// TIA Portal project "Voltra_Nord" (V21)

(* hardware
DEVICE "ET 200SP station_1"  ET 200SP-Station
   slot 0: "Rack_0"  Rack  6ES5 710-8MAx1
   slot 1: "Volta_Nord"  CPU 1510SP-1 PN  6ES7 510-1DK03-0AB0  V4.0
      slot 32768: "PROFINET interface_1"  X1
         slot 32771: "Port_3"  X1 P3
   slot 2: "CM PtP_1"  CM PtP  6ES7 137-6AA01-0BA0  V2.0
      slot 1: "CM PtP_1"  CM PtP Sub
   slot 3: "AI 8xRTD/TC 2-wire HF_1"  AI 8xRTD/TC 2-wire HF  6ES7 134-6JF00-0CA1  V2.1
      slot 1: "AI 8xRTD/TC 2-wire HF_1"  AI 8xRTD/TC 2-wire HF
   slot 4: "AI 8xRTD/TC 2-wire HF_2"  AI 8xRTD/TC 2-wire HF  6ES7 134-6JF00-0CA1  V2.1
      slot 1: "AI 8xRTD/TC 2-wire HF_2"  AI 8xRTD/TC 2-wire HF
   slot 5: "AI 8xI 2-/4-wire BA_1"  AI 8xI 2-,4-wire BA  6ES7 134-6GF00-0AA1  V1.0
      slot 1: "AI 8xI 2-/4-wire BA_1"  AI 8xI 2-,4-wire BA
   slot 6: "AI 8xI 2-/4-wire BA_2"  AI 8xI 2-,4-wire BA  6ES7 134-6GF00-0AA1  V1.0
      slot 1: "AI 8xI 2-/4-wire BA_2"  AI 8xI 2-,4-wire BA
   slot 7: "AQ 4xU/I ST_1"  AQ 4xU/I ST  6ES7 135-6HD00-0BA1  V1.1
      slot 1: "AQ 4xU/I ST_1"  AQ 4xU/I ST
   slot 8: "DI 16x24VDC ST_1"  DI 16x24VDC ST  6ES7 131-6BH01-0BA0  V0.0
      slot 1: "DI 16x24VDC ST_1"  DI 16x24VDC ST
   slot 9: "DI 16x24VDC ST_2"  DI 16x24VDC ST  6ES7 131-6BH01-0BA0  V0.0
      slot 1: "DI 16x24VDC ST_2"  DI 16x24VDC ST
   slot 10: "DI 16x24VDC ST_3"  DI 16x24VDC ST  6ES7 131-6BH01-0BA0  V0.0
      slot 1: "DI 16x24VDC ST_3"  DI 16x24VDC ST
   slot 11: "DQ 16x24VDC/0.5A BA_1"  DQ 16x24VDC/0.5A BA  6ES7 132-6BH00-0AA0  V0.0
      slot 1: "DQ 16x24VDC/0.5A BA_1"  DQ 16x24VDC/0.5A BA
   slot 12: "DQ 16x24VDC/0.5A BA_2"  DQ 16x24VDC/0.5A BA  6ES7 132-6BH00-0AA0  V0.0
      slot 1: "DQ 16x24VDC/0.5A BA_2"  DQ 16x24VDC/0.5A BA
   slot 13: "DQ 16x24VDC/0.5A BA_3"  DQ 16x24VDC/0.5A BA  6ES7 132-6BH00-0AA0  V0.0
      slot 1: "DQ 16x24VDC/0.5A BA_3"  DQ 16x24VDC/0.5A BA
   slot 14: "Server module_1"  Server module  6ES7 193-6PA00-0AA0  V1.2
      slot 1: "Server module_1"  Server module
   slot 127: "BA 2xRJ45"  BA 2xRJ45  6ES7 193-6AR00-0AA0  V0.0
      slot 32769: "Port_1"  X1 P1  6ES7 193-6AR00-0AA0
      slot 32770: "Port_2"  X1 P2  6ES7 193-6AR00-0AA0
*)

// ===== PLC "Volta_Nord"  CPU 1510SP-1 PN =====

VAR_GLOBAL   // PLC tag table "Default tag table"
   "Tag_1" AT %M100.0 : Bool;
   "System_Byte" AT %MB1 : Byte;
   "FirstScan" AT %M1.0 : Bool;
   "DiagStatusUpdate" AT %M1.1 : Bool;
   "AlwaysTRUE" AT %M1.2 : Bool;
   "AlwaysFALSE" AT %M1.3 : Bool;
   "Clock_Byte" AT %MB0 : Byte;
   "Clock_10Hz" AT %M0.0 : Bool;
   "Clock_5Hz" AT %M0.1 : Bool;
   "Clock_2.5Hz" AT %M0.2 : Bool;
   "Clock_2Hz" AT %M0.3 : Bool;
   "Clock_1.25Hz" AT %M0.4 : Bool;
   "Clock_1Hz" AT %M0.5 : Bool;
   "Clock_0.625Hz" AT %M0.6 : Bool;
   "Clock_0.5Hz" AT %M0.7 : Bool;
END_VAR

VAR_GLOBAL   // PLC tag table "RTD"
   "rM1OilTemp_C" AT %IW8 : Int;
   "rM1SuctionTemp_C" AT %IW10 : Int;
   "rM1DischargeTemp_C" AT %IW12 : Int;
   "rM2OilTemp_C" AT %IW14 : Int;
   "rM2SuctionTemp_C" AT %IW16 : Int;
   "rM2DischargeTemp_C" AT %IW18 : Int;
   "rM1EvapWaterOutTemp_C" AT %IW24 : Int;
   "rM1EvapWaterInTemp_C" AT %IW26 : Int;
   "rM1CondWaterOutTemp_C" AT %IW28 : Int;
   "rM1CondWaterInTemp_C" AT %IW30 : Int;
   "rM2EvapWaterOutTemp_C" AT %IW32 : Int;
   "rM2EvapWaterInTemp_C" AT %IW34 : Int;
   "rM2CondWaterOutTemp_C" AT %IW36 : Int;
   "rM2CondWaterInTemp_C" AT %IW38 : Int;
   "rm1OilTemp2_C" AT %IW20 : Int;
   "rm2OilTemp2_C" AT %IW22 : Int;
END_VAR

VAR_GLOBAL   // PLC tag table "AI"
   "rM1LiquidLevel_pct" AT %IW40 : Int;
   "rM1Pdis_bar" AT %IW42 : Int;
   "rM1Psuc_bar" AT %IW44 : Int;
   "rM1ViValvePos_pct" AT %IW46 : Int;
   "rM1ExtSetpointInput_C" AT %IW48 : Int;   // 9-10 klemes
   "rM2LiquidLevel_pct" AT %IW50 : Int;
   "rM2Pdis_bar" AT %IW52 : Int;
   "rM2Psuc_bar" AT %IW54 : Int;
   "rM2ExtSetpointInput_C" AT %IW58 : Int;   // 19-20 klemens
   "rM2ViValvePos_pct" AT %IW56 : Int;
   "AI_Rezerve1" AT %IW60 : Int;
   "AI_Rezerve2" AT %IW62 : Int;
   "AI_Rezerve3" AT %IW64 : Int;
   "AI_Rezerve4" AT %IW66 : Int;
   "AI_Rezerve5" AT %IW68 : Int;
   "AI_Rezerve6" AT %IW70 : Int;
END_VAR

VAR_GLOBAL   // PLC tag table "AQ"
   "rM1CompFreqRefOut_Hz" AT %QW0 : Int;
   "rM1ViValveCmd_pct" AT %QW2 : Int;
   "rM2CompFreqRefOut_Hz" AT %QW4 : Int;
   "rM2ViValveCmd_pct" AT %QW6 : Int;
END_VAR

VAR_GLOBAL   // PLC tag table "DI"
   "xPhaseProtectionRelaySig" AT %I72.0 : Bool;
   "xSafetySignal" AT %I72.1 : Bool;
   "xEmgStop" AT %I72.2 : Bool;
   "xM1EvapMotRunning" AT %I72.3 : Bool;
   "xM1CondenserMotRunning" AT %I72.4 : Bool;
   "xM1ExhaustFanRunning" AT %I72.5 : Bool;
   "xM1CompDriverRunnig" AT %I72.6 : Bool;
   "xM1CompDriverFault" AT %I72.7 : Bool;
   "xM1LiquidLowLevelSw" AT %I73.0 : Bool;
   "xM1LiquidHighLevelSw" AT %I73.1 : Bool;
   "xM2EvapMotRunning" AT %I73.2 : Bool;
   "xM2CondenserMotRunning" AT %I73.3 : Bool;
   "xM2ExhaustFanRunning" AT %I73.4 : Bool;
   "xM2CompDriverRunnig" AT %I73.5 : Bool;
   "xM2CompDriverFault" AT %I73.6 : Bool;
   "xM2LiquidLowLevelSw" AT %I73.7 : Bool;
   "xM2LiquidHighLevelSw" AT %I74.0 : Bool;
   "xM1OilFlowSw" AT %I74.1 : Bool;
   "xM1HighPressureSw" AT %I74.2 : Bool;
   "xM1LowPressureSw" AT %I74.3 : Bool;
   "xM1OilTankLowLevelSw" AT %I74.4 : Bool;
   "xM2OilFlowSw" AT %I74.5 : Bool;
   "xM2HighPressureSw" AT %I74.6 : Bool;
   "xM2LowPressureSw" AT %I74.7 : Bool;
   "xM2OilTankLowLevelSw" AT %I75.0 : Bool;
   "xM1BmsStartCoolEnableIn" AT %I75.1 : Bool;
   "xM1BmsStartHeatEnableIn" AT %I75.2 : Bool;
   "xM2BmsStartCoolEnableIn" AT %I75.3 : Bool;
   "xM2BmsStartHeatEnableIn" AT %I75.4 : Bool;
   "xM1EvapFlowSw" AT %I75.5 : Bool;
   "xM2EvapFlowSw" AT %I75.6 : Bool;
   "xM1CondenFlowSw" AT %I75.7 : Bool;
   "xM2CondenFlowSw" AT %I76.0 : Bool;
   "xM1OilHighLevelSwitch" AT %I76.1 : Bool;
   "xM2OilHighLevelSwitch" AT %I76.2 : Bool;
   "xM1GasFault" AT %I76.3 : Bool;
   "xM2GasFault" AT %I76.4 : Bool;
   "xM1CompThermalFault" AT %I76.5 : Bool;
   "xM2CompThermalFault" AT %I76.6 : Bool;
   "xM1HeaterRunnig" AT %I76.7 : Bool;
   "xM2HeaterRunnig" AT %I77.0 : Bool;
   "DI_Rezerve3" AT %I77.1 : Bool;
   "DI_Rezerve4" AT %I77.2 : Bool;
   "DI_Rezerve5" AT %I77.3 : Bool;
   "DI_Rezerve6" AT %I77.4 : Bool;
   "DI_Rezerve7" AT %I77.5 : Bool;
   "DI_Rezerve8" AT %I77.6 : Bool;
   "DI_Rezerve9" AT %I77.7 : Bool;
END_VAR

VAR_GLOBAL   // PLC tag table "DQ"
   "xM1EvapPumpCmd" AT %Q8.0 : Bool;
   "xM1CondPumpCmd" AT %Q8.1 : Bool;
   "xM1ExhaustFanCmd" AT %Q8.2 : Bool;
   "xM1CompRunCmd" AT %Q8.3 : Bool;
   "xM1TwoWayValveCmd" AT %Q8.4 : Bool;
   "xM1MvsEnableCmd1" AT %Q8.5 : Bool;   // 24v dc inildi panoda
   "xM1SystemOnRelayCmd" AT %Q8.6 : Bool;
   "xM1FaultRelayCmd" AT %Q8.7 : Bool;
   "xM1OilInletSolValve1Cmd" AT %Q9.0 : Bool;
   "xM1OilITempValve" AT %Q9.1 : Bool;
   "xM1OilReturnValve1" AT %Q9.2 : Bool;
   "xM1OilReturnValve2" AT %Q9.3 : Bool;
   "xM1StartLampCmd" AT %Q9.4 : Bool;
   "xM1FaultLampCmd" AT %Q9.5 : Bool;
   "xM1StopLampCmd" AT %Q9.6 : Bool;
   "xM2EvapPumpCmd" AT %Q9.7 : Bool;
   "xM2CondPumpCmd" AT %Q10.0 : Bool;
   "xM2ExhaustFanCmd" AT %Q10.1 : Bool;
   "xM2CompRunCmd" AT %Q10.2 : Bool;
   "xM2TwoWayValveCmd" AT %Q10.3 : Bool;
   "xM2MvsEnableCmd1" AT %Q10.4 : Bool;
   "xM2SystemOnRelayCmd" AT %Q10.5 : Bool;
   "xM2FaultRelayCmd" AT %Q10.6 : Bool;
   "xM2OillInletSolValve1Cmd" AT %Q10.7 : Bool;
   "xM2OilITempValve" AT %Q11.0 : Bool;
   "xM2OilReturnValve1" AT %Q11.1 : Bool;
   "xM2OilReturnValve2" AT %Q11.2 : Bool;
   "xM2StartLampCmd" AT %Q11.3 : Bool;
   "xM2FaultLampCmd" AT %Q11.4 : Bool;
   "xM2StopLampCmd" AT %Q11.5 : Bool;
   "xM1OilFlowValve" AT %Q11.6 : Bool;   // ICFE20H Slenoid Valve
   "xM2OilFlowValve" AT %Q11.7 : Bool;   // ICFE20H Slenoid Valve
   "xM1OilHeater" AT %Q12.0 : Bool;
   "xM2OilHeater" AT %Q12.1 : Bool;
   "xM1MvsEnableCmd2" AT %Q12.2 : Bool;
   "xM2MvsEnableCmd2" AT %Q12.3 : Bool;
   "DQ_Rezerve1" AT %Q12.4 : Bool;   // 220V AC PANOYA İNİLDİ
   "DQ_Rezerve2" AT %Q12.5 : Bool;   // 220V AC PANOYA İNİLDİ
   "DQ_Rezerve3" AT %Q12.6 : Bool;   // 220V AC PANOYA İNİLDİ
   "DQ_Rezerve4" AT %Q12.7 : Bool;   // 220V AC PANOYA İNİLDİ
   "DQ_Rezerve5" AT %Q13.0 : Bool;   // KURU KONTAK İNİLDİ
   "DQ_Rezerve6" AT %Q13.1 : Bool;   // KURU KONTAK İNİLDİ
   "DQ_Rezerve7" AT %Q13.2 : Bool;
   "DQ_Rezerve8" AT %Q13.3 : Bool;
   "DQ_Rezerve9" AT %Q13.4 : Bool;
   "DQ_Rezerve10" AT %Q13.5 : Bool;
   "DQ_Rezerve11" AT %Q13.6 : Bool;
   "DQ_Rezerve12" AT %Q13.7 : Bool;
END_VAR

DATA_BLOCK "AuxOutput"   // DB24
{ S7_Optimized_Access := 'TRUE' }
VERSION : 0.1
   VAR
      m1OilTempSelenoid : Bool;   // Makine 1 5 numara yağ soğutucusunun 25 numaralı valfinin çalışması için
      m2OilTempSelenoid : Bool;   // Makine 2 5 numara yağ soğutucusunun 25 numaralı valfinin çalışması için
      m1EvapOilValve3 : Bool;   // Makine 1 24 numaralı ekipman 1. selenoid valfi
      m1EvapOilValve4 : Bool;   // Makine 1 24 numaralı ekipman 2. selenoid valfi
      m2EvapOilValve3 : Bool;
      m2EvapOilValve4 : Bool;
   END_VAR
BEGIN
END_DATA_BLOCK

DATA_BLOCK "Alarm_DB"   // DB31
{ S7_Optimized_Access := 'FALSE' }
VERSION : 0.1
   VAR
      ALM_m1DischargeHighPressure : Bool;
      ALM_m2DischargeHighPressure : Bool;
      ALM_m1DischargeLowPressure : Bool;
      ALM_m2DischargeLowPressure : Bool;
      ALM_m1KrıwanThermalFault : Bool;
      ALM_m2KrıwanThermalFault : Bool;
      ALM_m1OilFlowFault : Bool;
      ALM_m2OilFlowFault : Bool;
      ALM_m1CondensFlowFault : Bool;
      ALM_m2CondensFlowFault : Bool;
      ALM_m1EvapFlowFault : Bool;
      ALM_m2EvapFlowFault : Bool;
      ALM_m1EvapLiquidHighLevelFault : Bool;
      ALM_m2EvapLiquidHighLevelFault : Bool;
      ALM_m1EvapLiquidLowLevelFault : Bool;
      ALM_m2EvapLiquidLowLevelFault : Bool;
      ALM_m1OilTempHighFault : Bool;
      ALM_m2OilTempHighFault : Bool;
      ALM_m1OilTempHighHighFault : Bool;
      ALM_m2OilTempHighHighFault : Bool;
      ALM_m1EvapFlowWarning : Bool;
      ALM_m2EvapFlowWarning : Bool;
      ALM_m1CondensFlowWarning : Bool;
      ALM_m2CondensFlowWarning : Bool;
      ALM_m1NH3Fault : Bool;
      ALM_m2NH3Fault : Bool;
      ALM_m1CompInvFault : Bool;
      ALM_m2CompInvFault : Bool;
      ALM_PhaseProtectionRelayFault : Bool;
      ALM_SafetyFault : Bool;
      ALM_EmgFault : Bool;
      ALM_m1CompDriverFault : Bool;
      ALM_m2CompDriverFault : Bool;
      ALM_m1CondensMotorFault : Bool;
      ALM_m2CondensMotorFault_1 : Bool;
      ALM_m1EvapMotorFault : Bool;
      ALM_m2EvapMotorFault : Bool;
   END_VAR
BEGIN
END_DATA_BLOCK

DATA_BLOCK "General_DB"   // DB32
{ S7_Optimized_Access := 'FALSE' }
VERSION : 0.1
   VAR
      m1FlowOilAlarmEnable : Bool;
      m2FlowOilAlarmEnable : Bool;
      m1CondensFlowAlarmEnable : Bool;
      m2CondensFlowAlarmEnable : Bool;
      m1EvapFlowAlarmEnable : Bool;
      m2EvapFlowAlarmEnable : Bool;
      m1EvapLiquidHighLevelEnable : Bool;
      m2EvapLiquidHighLevelEnable : Bool;
      m1EvapLiquidLowLevelEnable : Bool;
      m2EvapLiquidLowLevelEnable : Bool;
      m1OilTempHighHighEnable : Bool;
      m2OilTempHighHighEnable : Bool;
      m1DischargeTempHighEnable : Bool;
      m2DischargeTempHighEnable : Bool;
      m1DischargeTempHighHighEnable : Bool;
      m2DischargeTempHighHighEnable : Bool;
      m1EvapFlowWarningEnable : Bool;
      m2EvapFlowWarningEnable : Bool;
      m1CondensFlowWarningEnable : Bool;
      m2CondensFlowWarningEnable : Bool;
      m1OilTempHighEnable : Bool;
      m2OilTempHighEnable : Bool;
      m1OilTempOk : Bool;
      m2OilTempOk : Bool;
      m1Status : Int;
      m2Status : Int;
      m1StartCoolling : Bool;
      m1StartHeating : Bool;
   END_VAR
BEGIN
END_DATA_BLOCK

DATA_BLOCK "PidVar_DB"   // DB41
{ S7_Optimized_Access := 'FALSE' }
VERSION : 0.1
   VAR
      m1PidSetPoint : Real;
      m1ManualEnable : Bool;
      m1ManualValue : Real;
      m1ErrorAck : Bool;
      m1Reset : Bool;
      m1ModeActivate : Bool;
      m1Mode : Int;
      m2PidSetPoint : Real;
      m2ManualEnable : Bool;
      m2ManualValue : Real;
      m2ErrorAck : Bool;
      m2Reset : Bool;
      m2ModeActivate : Bool;
      m2Mode : Int;
      m1LiquidLevelSet : Real;
      m1ExpManEnable : Bool;
      m1ExpManValue : Real;
      m1LiquidErrorAck : Bool;
      m1LiquidPidReset : Bool;
      m1LiquidModeActive : Bool;
      m1LiquidModePid : Int;
      m2LiquidLevelSet : Real;
      m2ExpManEnable : Bool;
      m2ExpManValue : Real;
      m2LiquidErrorAck : Bool;
      m2LiquidPidReset : Bool;
      m2LiquidModeActive : Bool;
      m2LiquidModePid : Int;
   END_VAR
BEGIN
END_DATA_BLOCK

// folder: Hmi

DATA_BLOCK "Pressure_Scale"   // DB2
{ S7_Optimized_Access := 'FALSE' }
VERSION : 0.1
   VAR
      M1PdisOut_Max : Real;
      M1PdisOut_Min : Real;
      M1PdisIn_Max : Real;
      M1PdisIn_Min : Real;
      M1PdisAlpha : Real := 1.0;
      M2PdisOut_Max : Real;
      M2PdisOut_Min : Real;
      M2PdisIn_Max : Real;
      M2PdisIn_Min : Real;
      M2PdisAlpha : Real := 1.0;
      M1PSecOut_Max : Real;
      M1PSecOut_Min : Real;
      M1PSecIn_Max : Real;
      M1PSecIn_Min : Real;
      M1PSecAlpha : Real := 1.0;
      M2PSecOut_Max : Real;
      M2PSecOut_Min : Real;
      M2PSecIn_Max : Real;
      M2PSecIn_Min : Real;
      M2PSecAlpha : Real := 1.0;
   END_VAR
BEGIN
END_DATA_BLOCK

DATA_BLOCK "Liquid_Level"   // DB6
{ S7_Optimized_Access := 'FALSE' }
VERSION : 0.1
   VAR
      M1LiquidLvlOut_Max : Real;
      M1LiquidLvlOut_Min : Real;
      M1LiquidLvlIn_Max : Real;
      M1LiquidLvlIn_Min : Real;
      M1LiquidLvlAlpha : Real;
      M2LiquidLvlOut_Max : Real;
      M2LiquidLvlOut_Min : Real;
      M2LiquidLvlIn_Max : Real;
      M2LiquidLvlIn_Min : Real;
      M2LiquidLvlAlpha : Real;
   END_VAR
BEGIN
END_DATA_BLOCK

DATA_BLOCK "HMI"   // DB23
{ S7_Optimized_Access := 'FALSE' }
VERSION : 0.1
   VAR
      rM1OilTempHis : Real;
      rM1OilTempSet : Real;
      rM2OilTempHis : Real;
      rM2OilTempSet : Real;
      tM1EvapOilHisTime : Time;   // M1 24 numaralı ekipman sensörünün filtresi için koyuldu
      tM1EvapOilDischargeTime : Time;   // M1 24 numaralı ekipmanın basınç hattının valfinin açık kalma süresi
      tM1EvapOilDischargeWaitTime : Time;   // M1 24 numaralı ekipmanın basınç hattının valfinin bekleme süresi
      tM2EvapOilHisTime : Time;
      tM2EvapOilDischargeTime : Time;
      tM2EvapOilDischargeWaitTime : Time;
      m1SetDischargeHighPressure : Real;
      m2SetDischargeHighPressure : Real;
      m1SetDischargeLowPressure : Real;
      m2SetDischargeLowPressure : Real;
      m1OilTempHighHighSet : Real;
      m2OilTempHighHighSet : Real;
      m1DischargeTempHighSet : Real;
      m2DischargeTempHighSet : Real;
      m1DischargeTempHighHighSet : Real;
      m2DischargeTempHighHighSet : Real;
      m1OilTempHighSet : Real;
      m2OilTempHighSet : Real;
      m1OilStartTempSet : Real;
      m2OilStartTempSet : Real;
      m1Status : Int;
      m1ExtValveScaleAlpha : Real := 1.0;
      m2ExtValveScaleAlpha : Real := 1.0;
   END_VAR
BEGIN
END_DATA_BLOCK

DATA_BLOCK "TempSet"   // DB39
{ S7_Optimized_Access := 'FALSE' }
VERSION : 0.1
   VAR
      m1TempSetOut_Max : Real;
      m1TempSetOut_Min : Real;
      m1TempSetIn_Max : Real;
      m1TempSetIn_Min : Real;
      m1TempSetAlpha : Real := 1.0;
      m2TempSetOut_Max : Real;
      m2TempSetOut_Min : Real;
      m2TempSetIn_Max : Real;
      m2TempSetIn_Min : Real;
      m2TempSetAlpha : Real := 1.0;
   END_VAR
BEGIN
END_DATA_BLOCK

// folder: Scale_DB

DATA_BLOCK "M1Pdischarge"   // DB1
{ S7_Optimized_Access := 'TRUE' }
VERSION : 0.1
// stored: InstanceOfName Scale
"Scale"
BEGIN
END_DATA_BLOCK

DATA_BLOCK "M2Pdischarge"   // DB3
{ S7_Optimized_Access := 'TRUE' }
VERSION : 0.1
// stored: InstanceOfName Scale
"Scale"
BEGIN
END_DATA_BLOCK

DATA_BLOCK "M1PSec"   // DB4
{ S7_Optimized_Access := 'TRUE' }
VERSION : 0.1
// stored: InstanceOfName Scale
"Scale"
BEGIN
END_DATA_BLOCK

DATA_BLOCK "M2Psec"   // DB5
{ S7_Optimized_Access := 'TRUE' }
VERSION : 0.1
// stored: InstanceOfName Scale
"Scale"
BEGIN
END_DATA_BLOCK

DATA_BLOCK "M1LiquidLevel"   // DB7
{ S7_Optimized_Access := 'TRUE' }
VERSION : 0.1
// stored: InstanceOfName Scale
"Scale"
BEGIN
END_DATA_BLOCK

DATA_BLOCK "M2LiquidLevel"   // DB8
{ S7_Optimized_Access := 'TRUE' }
VERSION : 0.1
// stored: InstanceOfName Scale
"Scale"
BEGIN
END_DATA_BLOCK

DATA_BLOCK "m1Discharge_TT"   // DB9
{ S7_Optimized_Access := 'TRUE' }
VERSION : 0.1
// stored: InstanceOfName RTD
"RTD"
BEGIN
END_DATA_BLOCK

DATA_BLOCK "m2Discharge_TT"   // DB10
{ S7_Optimized_Access := 'TRUE' }
VERSION : 0.1
// stored: InstanceOfName RTD
"RTD"
BEGIN
END_DATA_BLOCK

DATA_BLOCK "m1Section_TT"   // DB11
{ S7_Optimized_Access := 'TRUE' }
VERSION : 0.1
// stored: InstanceOfName RTD
"RTD"
BEGIN
END_DATA_BLOCK

DATA_BLOCK "m2Section_TT"   // DB12
{ S7_Optimized_Access := 'TRUE' }
VERSION : 0.1
// stored: InstanceOfName RTD
"RTD"
BEGIN
END_DATA_BLOCK

DATA_BLOCK "m1Oil_TT"   // DB13
{ S7_Optimized_Access := 'TRUE' }
VERSION : 0.1
// stored: InstanceOfName RTD
"RTD"
BEGIN
END_DATA_BLOCK

DATA_BLOCK "m2Oil_TT"   // DB14
{ S7_Optimized_Access := 'TRUE' }
VERSION : 0.1
// stored: InstanceOfName RTD
"RTD"
BEGIN
END_DATA_BLOCK

DATA_BLOCK "m1EvapWatOut_TT"   // DB15
{ S7_Optimized_Access := 'TRUE' }
VERSION : 0.1
// stored: InstanceOfName RTD
"RTD"
BEGIN
END_DATA_BLOCK

DATA_BLOCK "m1EvapWatIn_TT"   // DB16
{ S7_Optimized_Access := 'TRUE' }
VERSION : 0.1
// stored: InstanceOfName RTD
"RTD"
BEGIN
END_DATA_BLOCK

DATA_BLOCK "m2EvapWatOut_TT"   // DB17
{ S7_Optimized_Access := 'TRUE' }
VERSION : 0.1
// stored: InstanceOfName RTD
"RTD"
BEGIN
END_DATA_BLOCK

DATA_BLOCK "m2EvapWatIn_TT"   // DB18
{ S7_Optimized_Access := 'TRUE' }
VERSION : 0.1
// stored: InstanceOfName RTD
"RTD"
BEGIN
END_DATA_BLOCK

DATA_BLOCK "m1ConWatOut_TT"   // DB19
{ S7_Optimized_Access := 'TRUE' }
VERSION : 0.1
// stored: InstanceOfName RTD
"RTD"
BEGIN
END_DATA_BLOCK

DATA_BLOCK "m1ConWatIn_TT"   // DB20
{ S7_Optimized_Access := 'TRUE' }
VERSION : 0.1
// stored: InstanceOfName RTD
"RTD"
BEGIN
END_DATA_BLOCK

DATA_BLOCK "m2ConWatOut_TT"   // DB21
{ S7_Optimized_Access := 'TRUE' }
VERSION : 0.1
// stored: InstanceOfName RTD
"RTD"
BEGIN
END_DATA_BLOCK

DATA_BLOCK "m2ConWatIn_TT"   // DB22
{ S7_Optimized_Access := 'TRUE' }
VERSION : 0.1
// stored: InstanceOfName RTD
"RTD"
BEGIN
END_DATA_BLOCK

DATA_BLOCK "m1TempSetScale"   // DB38
{ S7_Optimized_Access := 'TRUE' }
VERSION : 0.1
// stored: InstanceOfName Scale
"Scale"
BEGIN
END_DATA_BLOCK

DATA_BLOCK "m2TempSetScale"   // DB40
{ S7_Optimized_Access := 'TRUE' }
VERSION : 0.1
// stored: InstanceOfName Scale
"Scale"
BEGIN
END_DATA_BLOCK

DATA_BLOCK "m1ExtValvePoz"   // DB45
{ S7_Optimized_Access := 'TRUE' }
VERSION : 0.1
// stored: InstanceOfName Scale
"Scale"
BEGIN
END_DATA_BLOCK

DATA_BLOCK "m2ExtValvePoz"   // DB46
{ S7_Optimized_Access := 'TRUE' }
VERSION : 0.1
// stored: InstanceOfName Scale
"Scale"
BEGIN
END_DATA_BLOCK

// folder: System blocks/Program resources

DATA_BLOCK "m1EvapOilSenFilter_Time"   // DB25
{ S7_Optimized_Access := 'TRUE' }
AUTHOR : Simatic
FAMILY : IEC
NAME : IEC_TMR
VERSION : 1.0
// stored: InstanceOfName IEC_TIMER
"IEC_TIMER"
BEGIN
END_DATA_BLOCK

DATA_BLOCK "m1EvapOilValve4Run_Time"   // DB26
{ S7_Optimized_Access := 'TRUE' }
AUTHOR : Simatic
FAMILY : IEC
NAME : IEC_TMR
VERSION : 1.0
// stored: InstanceOfName IEC_TIMER
"IEC_TIMER"
BEGIN
END_DATA_BLOCK

DATA_BLOCK "m1EvapOilValve4Wait_Time"   // DB27
{ S7_Optimized_Access := 'TRUE' }
AUTHOR : Simatic
FAMILY : IEC
NAME : IEC_TMR
VERSION : 1.0
// stored: InstanceOfName IEC_TIMER
"IEC_TIMER"
BEGIN
END_DATA_BLOCK

DATA_BLOCK "m2EvapOilSenFilter_Time"   // DB28
{ S7_Optimized_Access := 'TRUE' }
AUTHOR : Simatic
FAMILY : IEC
NAME : IEC_TMR
VERSION : 1.0
// stored: InstanceOfName IEC_TIMER
"IEC_TIMER"
BEGIN
END_DATA_BLOCK

DATA_BLOCK "m2EvapOilValve4Run_Time"   // DB29
{ S7_Optimized_Access := 'TRUE' }
AUTHOR : Simatic
FAMILY : IEC
NAME : IEC_TMR
VERSION : 1.0
// stored: InstanceOfName IEC_TIMER
"IEC_TIMER"
BEGIN
END_DATA_BLOCK

DATA_BLOCK "m2EvapOilValve4Wait_Time"   // DB30
{ S7_Optimized_Access := 'TRUE' }
AUTHOR : Simatic
FAMILY : IEC
NAME : IEC_TMR
VERSION : 1.0
// stored: InstanceOfName IEC_TIMER
"IEC_TIMER"
BEGIN
END_DATA_BLOCK

DATA_BLOCK "m1CondensFlowFaultTime"   // DB33
{ S7_Optimized_Access := 'TRUE' }
AUTHOR : Simatic
FAMILY : IEC
NAME : IEC_TMR
VERSION : 1.0
// stored: InstanceOfName IEC_TIMER
"IEC_TIMER"
BEGIN
END_DATA_BLOCK

DATA_BLOCK "m2CondensFlowFaultTime"   // DB34
{ S7_Optimized_Access := 'TRUE' }
AUTHOR : Simatic
FAMILY : IEC
NAME : IEC_TMR
VERSION : 1.0
// stored: InstanceOfName IEC_TIMER
"IEC_TIMER"
BEGIN
END_DATA_BLOCK

DATA_BLOCK "m1EvapFlowFaultTime"   // DB35
{ S7_Optimized_Access := 'TRUE' }
AUTHOR : Simatic
FAMILY : IEC
NAME : IEC_TMR
VERSION : 1.0
// stored: InstanceOfName IEC_TIMER
"IEC_TIMER"
BEGIN
END_DATA_BLOCK

DATA_BLOCK "m2EvapFlowFaultTime"   // DB36
{ S7_Optimized_Access := 'TRUE' }
AUTHOR : Simatic
FAMILY : IEC
NAME : IEC_TMR
VERSION : 1.0
// stored: InstanceOfName IEC_TIMER
"IEC_TIMER"
BEGIN
END_DATA_BLOCK

// folder: (top level)

FUNCTION_BLOCK "RTD"   // FB1, SCL
{ S7_Optimized_Access := 'TRUE' }
VERSION : 0.1
   VAR_INPUT
      TempIn : Int;
   END_VAR
   VAR_OUTPUT
      Temp_O : Real;
   END_VAR
   VAR_TEMP
      TemDınt : DInt;
      TempReal : Real;
   END_VAR
BEGIN
   #TemDınt := INT_TO_DINT(#TempIn);
   #TempReal := DINT_TO_REAL(#TemDınt);
   #Temp_O := #TempReal / 10.0;
END_FUNCTION_BLOCK

FUNCTION_BLOCK "Scale"   // FB2, SCL
{ S7_Optimized_Access := 'TRUE' }
VERSION : 0.1
   VAR_INPUT
      Output_Max : Real;
      Output_Min : Real;
      Input_Max : Real;
      Input_Min : Real;
      Actual_Analog : Int;
   END_VAR
   VAR_OUTPUT
      filteredOutput : Real;
      ErrorAnalog : Bool;
   END_VAR
   VAR_IN_OUT
      alpha : Real;
   END_VAR
   VAR
      Sub_Value : Real;
      Source_Value : Real;
      Slope_Value : Real;
      Kx_Value : Real;
      Min_Slope_Value : Real;
      Ofset_Value : Real;
      scaledValue : Real;
      prevFilteredValue : Real;
      Actual_Analog_Real : Real;
   END_VAR
BEGIN
   #Actual_Analog_Real := INT_TO_REAL(#Actual_Analog);


   #Sub_Value := #Output_Max - #Output_Min;    //Skala edeceğimiz max ve min değer birbirinden çıkardık
   #Source_Value := #Input_Max - #Input_Min; //Analog değerin maksimum ve min değeri birbirinden çıkartıldı. 
   IF #Source_Value <> 0 THEN
       #Slope_Value := #Sub_Value / #Source_Value;
   END_IF;
   #Kx_Value := #Slope_Value * #Actual_Analog_Real;
   #Min_Slope_Value := #Slope_Value * #Input_Min;
   #Ofset_Value := #Output_Min - #Min_Slope_Value;
   #scaledValue := #Kx_Value + #Ofset_Value;
   IF #alpha <= 0.0 THEN
       #alpha := 0;
   ELSIF #alpha >= 1.0 THEN
       #alpha := 1;
   END_IF;

   #filteredOutput := #alpha * #scaledValue + (1 - #alpha) * #prevFilteredValue;
   #prevFilteredValue := #filteredOutput; // Yeni değeri sakla

   IF #Actual_Analog > 27648 THEN
       #ErrorAnalog := TRUE;
   END_IF;


   IF 0<#Actual_Analog AND 27468>=#Actual_Analog THEN
       #ErrorAnalog := FALSE;
   END_IF;
END_FUNCTION_BLOCK

FUNCTION "Analog" : Void   // FC1, LAD
{ S7_Optimized_Access := 'TRUE' }
VERSION : 0.1
BEGIN

REGION Network 1: M1 pressure discharge line PT transmitter scale
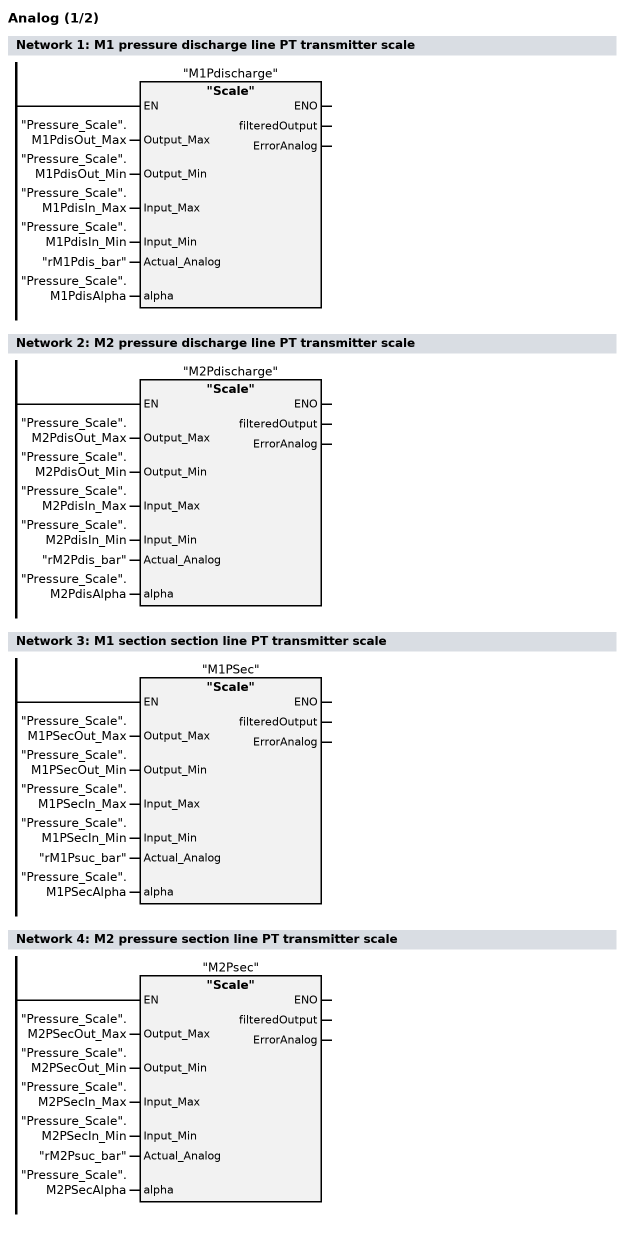
   RUNG wire#powerrail
      "M1Pdischarge"(Output_Max := "Pressure_Scale".M1PdisOut_Max, Output_Min := "Pressure_Scale".M1PdisOut_Min, Input_Max := "Pressure_Scale".M1PdisIn_Max, Input_Min := "Pressure_Scale".M1PdisIn_Min, Actual_Analog := "rM1Pdis_bar", alpha := "Pressure_Scale".M1PdisAlpha, filteredOutput =>, ErrorAnalog =>)
   END_RUNG
   // the same network as SCL:
   "M1Pdischarge"(Output_Max := "Pressure_Scale".M1PdisOut_Max,   // "Scale"
                  Output_Min := "Pressure_Scale".M1PdisOut_Min,
                  Input_Max := "Pressure_Scale".M1PdisIn_Max,
                  Input_Min := "Pressure_Scale".M1PdisIn_Min,
                  Actual_Analog := "rM1Pdis_bar",
                  alpha := "Pressure_Scale".M1PdisAlpha);
END_REGION

REGION Network 2: M2 pressure discharge line PT transmitter scale
   RUNG wire#powerrail
      "M2Pdischarge"(Output_Max := "Pressure_Scale".M2PdisOut_Max, Output_Min := "Pressure_Scale".M2PdisOut_Min, Input_Max := "Pressure_Scale".M2PdisIn_Max, Input_Min := "Pressure_Scale".M2PdisIn_Min, Actual_Analog := "rM2Pdis_bar", alpha := "Pressure_Scale".M2PdisAlpha, filteredOutput =>, ErrorAnalog =>)
   END_RUNG
   // the same network as SCL:
   "M2Pdischarge"(Output_Max := "Pressure_Scale".M2PdisOut_Max,   // "Scale"
                  Output_Min := "Pressure_Scale".M2PdisOut_Min,
                  Input_Max := "Pressure_Scale".M2PdisIn_Max,
                  Input_Min := "Pressure_Scale".M2PdisIn_Min,
                  Actual_Analog := "rM2Pdis_bar",
                  alpha := "Pressure_Scale".M2PdisAlpha);
END_REGION

REGION Network 3: M1 section section line PT transmitter scale
   RUNG wire#powerrail
      "M1PSec"(Output_Max := "Pressure_Scale".M1PSecOut_Max, Output_Min := "Pressure_Scale".M1PSecOut_Min, Input_Max := "Pressure_Scale".M1PSecIn_Max, Input_Min := "Pressure_Scale".M1PSecIn_Min, Actual_Analog := "rM1Psuc_bar", alpha := "Pressure_Scale".M1PSecAlpha, filteredOutput =>, ErrorAnalog =>)
   END_RUNG
   // the same network as SCL:
   "M1PSec"(Output_Max := "Pressure_Scale".M1PSecOut_Max,   // "Scale"
            Output_Min := "Pressure_Scale".M1PSecOut_Min,
            Input_Max := "Pressure_Scale".M1PSecIn_Max,
            Input_Min := "Pressure_Scale".M1PSecIn_Min,
            Actual_Analog := "rM1Psuc_bar",
            alpha := "Pressure_Scale".M1PSecAlpha);
END_REGION

REGION Network 4: M2 pressure section line PT transmitter scale
   RUNG wire#powerrail
      "M2Psec"(Output_Max := "Pressure_Scale".M2PSecOut_Max, Output_Min := "Pressure_Scale".M2PSecOut_Min, Input_Max := "Pressure_Scale".M2PSecIn_Max, Input_Min := "Pressure_Scale".M2PSecIn_Min, Actual_Analog := "rM2Psuc_bar", alpha := "Pressure_Scale".M2PSecAlpha, filteredOutput =>, ErrorAnalog =>)
   END_RUNG
   // the same network as SCL:
   "M2Psec"(Output_Max := "Pressure_Scale".M2PSecOut_Max,   // "Scale"
            Output_Min := "Pressure_Scale".M2PSecOut_Min,
            Input_Max := "Pressure_Scale".M2PSecIn_Max,
            Input_Min := "Pressure_Scale".M2PSecIn_Min,
            Actual_Analog := "rM2Psuc_bar",
            alpha := "Pressure_Scale".M2PSecAlpha);
END_REGION

REGION Network 5: M1 Liquid Level Switch
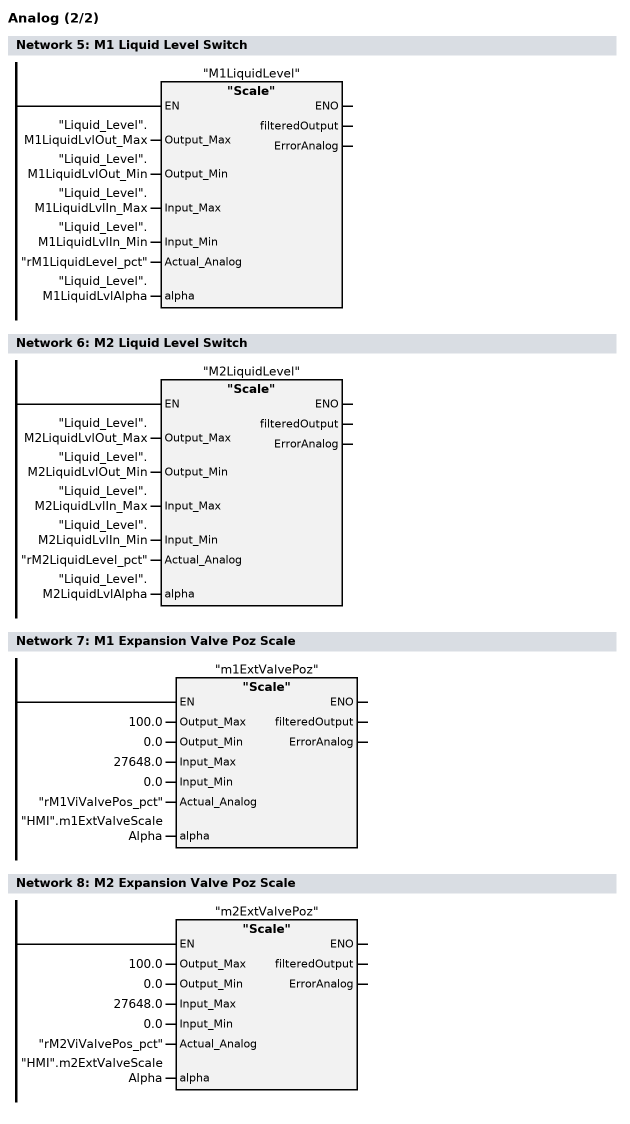
   RUNG wire#powerrail
      "M1LiquidLevel"(Output_Max := "Liquid_Level".M1LiquidLvlOut_Max, Output_Min := "Liquid_Level".M1LiquidLvlOut_Min, Input_Max := "Liquid_Level".M1LiquidLvlIn_Max, Input_Min := "Liquid_Level".M1LiquidLvlIn_Min, Actual_Analog := "rM1LiquidLevel_pct", alpha := "Liquid_Level".M1LiquidLvlAlpha, filteredOutput =>, ErrorAnalog =>)
   END_RUNG
   // the same network as SCL:
   "M1LiquidLevel"(Output_Max := "Liquid_Level".M1LiquidLvlOut_Max,   // "Scale"
                   Output_Min := "Liquid_Level".M1LiquidLvlOut_Min,
                   Input_Max := "Liquid_Level".M1LiquidLvlIn_Max,
                   Input_Min := "Liquid_Level".M1LiquidLvlIn_Min,
                   Actual_Analog := "rM1LiquidLevel_pct",
                   alpha := "Liquid_Level".M1LiquidLvlAlpha);
END_REGION

REGION Network 6: M2 Liquid Level Switch
   RUNG wire#powerrail
      "M2LiquidLevel"(Output_Max := "Liquid_Level".M2LiquidLvlOut_Max, Output_Min := "Liquid_Level".M2LiquidLvlOut_Min, Input_Max := "Liquid_Level".M2LiquidLvlIn_Max, Input_Min := "Liquid_Level".M2LiquidLvlIn_Min, Actual_Analog := "rM2LiquidLevel_pct", alpha := "Liquid_Level".M2LiquidLvlAlpha, filteredOutput =>, ErrorAnalog =>)
   END_RUNG
   // the same network as SCL:
   "M2LiquidLevel"(Output_Max := "Liquid_Level".M2LiquidLvlOut_Max,   // "Scale"
                   Output_Min := "Liquid_Level".M2LiquidLvlOut_Min,
                   Input_Max := "Liquid_Level".M2LiquidLvlIn_Max,
                   Input_Min := "Liquid_Level".M2LiquidLvlIn_Min,
                   Actual_Analog := "rM2LiquidLevel_pct",
                   alpha := "Liquid_Level".M2LiquidLvlAlpha);
END_REGION

REGION Network 7: M1 Expansion Valve Poz Scale
   RUNG wire#powerrail
      "m1ExtValvePoz"(Output_Max := 100.0, Output_Min := 0.0, Input_Max := 27648.0, Input_Min := 0.0, Actual_Analog := "rM1ViValvePos_pct", alpha := "HMI".m1ExtValveScaleAlpha, filteredOutput =>, ErrorAnalog =>)
   END_RUNG
   // the same network as SCL:
   "m1ExtValvePoz"(Output_Max := 100.0,   // "Scale"
                   Output_Min := 0.0,
                   Input_Max := 27648.0,
                   Input_Min := 0.0,
                   Actual_Analog := "rM1ViValvePos_pct",
                   alpha := "HMI".m1ExtValveScaleAlpha);
END_REGION

REGION Network 8: M2 Expansion Valve Poz Scale
   RUNG wire#powerrail
      "m2ExtValvePoz"(Output_Max := 100.0, Output_Min := 0.0, Input_Max := 27648.0, Input_Min := 0.0, Actual_Analog := "rM2ViValvePos_pct", alpha := "HMI".m2ExtValveScaleAlpha, filteredOutput =>, ErrorAnalog =>)
   END_RUNG
   // the same network as SCL:
   "m2ExtValvePoz"(Output_Max := 100.0,   // "Scale"
                   Output_Min := 0.0,
                   Input_Max := 27648.0,
                   Input_Min := 0.0,
                   Actual_Analog := "rM2ViValvePos_pct",
                   alpha := "HMI".m2ExtValveScaleAlpha);
END_REGION
END_FUNCTION

FUNCTION "Temprature" : Void   // FC2, LAD
{ S7_Optimized_Access := 'TRUE' }
VERSION : 0.1
BEGIN

REGION Network 1: M1 Discharge Temperature
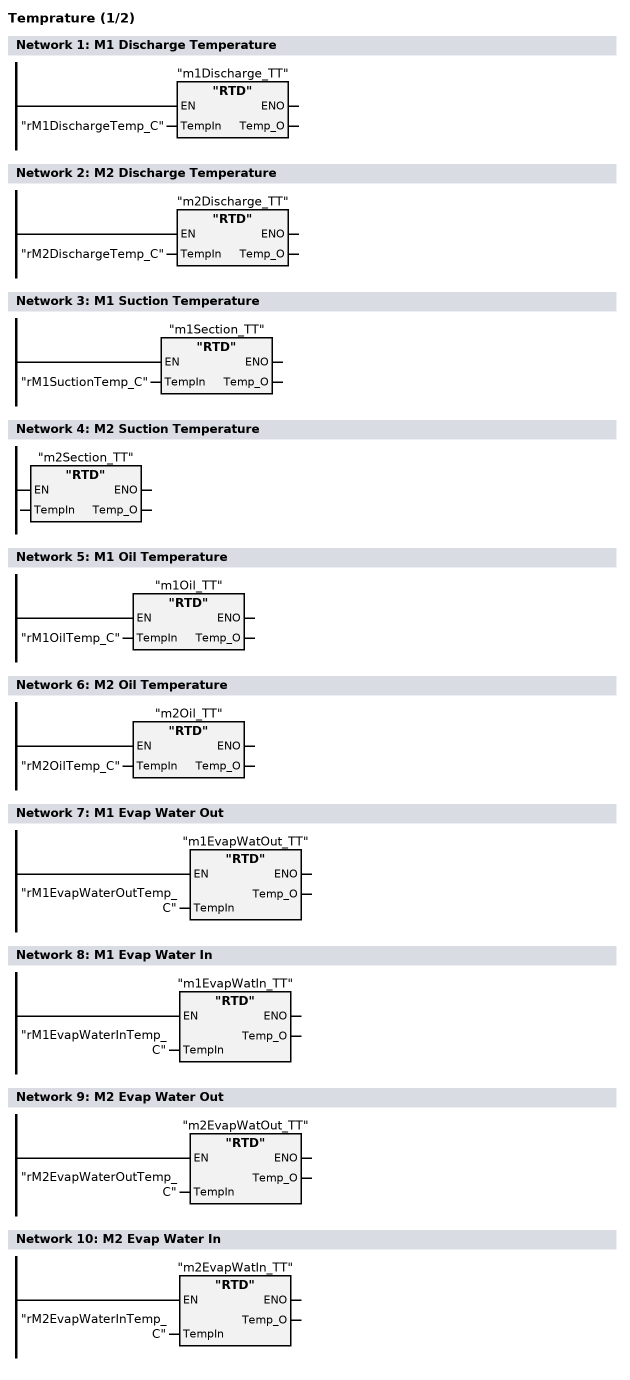
   RUNG wire#powerrail
      "m1Discharge_TT"(TempIn := "rM1DischargeTemp_C", Temp_O =>)
   END_RUNG
   // the same network as SCL:
   "m1Discharge_TT"(TempIn := "rM1DischargeTemp_C");   // "RTD"
END_REGION

REGION Network 2: M2 Discharge Temperature
   RUNG wire#powerrail
      "m2Discharge_TT"(TempIn := "rM2DischargeTemp_C", Temp_O =>)
   END_RUNG
   // the same network as SCL:
   "m2Discharge_TT"(TempIn := "rM2DischargeTemp_C");   // "RTD"
END_REGION

REGION Network 3: M1 Suction Temperature
   RUNG wire#powerrail
      "m1Section_TT"(TempIn := "rM1SuctionTemp_C", Temp_O =>)
   END_RUNG
   // the same network as SCL:
   "m1Section_TT"(TempIn := "rM1SuctionTemp_C");   // "RTD"
END_REGION

REGION Network 4: M2 Suction Temperature
   RUNG wire#powerrail
      "m2Section_TT"(TempIn :=, Temp_O =>)
   END_RUNG
   // the same network as SCL:
   "m2Section_TT"();   // "RTD"
END_REGION

REGION Network 5: M1 Oil Temperature
   RUNG wire#powerrail
      "m1Oil_TT"(TempIn := "rM1OilTemp_C", Temp_O =>)
   END_RUNG
   // the same network as SCL:
   "m1Oil_TT"(TempIn := "rM1OilTemp_C");   // "RTD"
END_REGION

REGION Network 6: M2 Oil Temperature
   RUNG wire#powerrail
      "m2Oil_TT"(TempIn := "rM2OilTemp_C", Temp_O =>)
   END_RUNG
   // the same network as SCL:
   "m2Oil_TT"(TempIn := "rM2OilTemp_C");   // "RTD"
END_REGION

REGION Network 7: M1 Evap Water Out
   RUNG wire#powerrail
      "m1EvapWatOut_TT"(TempIn := "rM1EvapWaterOutTemp_C", Temp_O =>)
   END_RUNG
   // the same network as SCL:
   "m1EvapWatOut_TT"(TempIn := "rM1EvapWaterOutTemp_C");   // "RTD"
END_REGION

REGION Network 8: M1 Evap Water In
   RUNG wire#powerrail
      "m1EvapWatIn_TT"(TempIn := "rM1EvapWaterInTemp_C", Temp_O =>)
   END_RUNG
   // the same network as SCL:
   "m1EvapWatIn_TT"(TempIn := "rM1EvapWaterInTemp_C");   // "RTD"
END_REGION

REGION Network 9: M2 Evap Water Out
   RUNG wire#powerrail
      "m2EvapWatOut_TT"(TempIn := "rM2EvapWaterOutTemp_C", Temp_O =>)
   END_RUNG
   // the same network as SCL:
   "m2EvapWatOut_TT"(TempIn := "rM2EvapWaterOutTemp_C");   // "RTD"
END_REGION

REGION Network 10: M2 Evap Water In
   RUNG wire#powerrail
      "m2EvapWatIn_TT"(TempIn := "rM2EvapWaterInTemp_C", Temp_O =>)
   END_RUNG
   // the same network as SCL:
   "m2EvapWatIn_TT"(TempIn := "rM2EvapWaterInTemp_C");   // "RTD"
END_REGION

REGION Network 11: M1 Condenser Water Out
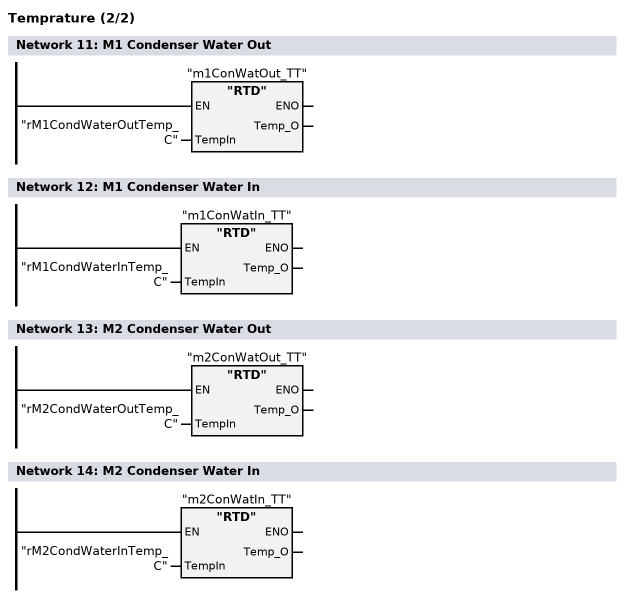
   RUNG wire#powerrail
      "m1ConWatOut_TT"(TempIn := "rM1CondWaterOutTemp_C", Temp_O =>)
   END_RUNG
   // the same network as SCL:
   "m1ConWatOut_TT"(TempIn := "rM1CondWaterOutTemp_C");   // "RTD"
END_REGION

REGION Network 12: M1 Condenser Water In
   RUNG wire#powerrail
      "m1ConWatIn_TT"(TempIn := "rM1CondWaterInTemp_C", Temp_O =>)
   END_RUNG
   // the same network as SCL:
   "m1ConWatIn_TT"(TempIn := "rM1CondWaterInTemp_C");   // "RTD"
END_REGION

REGION Network 13: M2 Condenser Water Out
   RUNG wire#powerrail
      "m2ConWatOut_TT"(TempIn := "rM2CondWaterOutTemp_C", Temp_O =>)
   END_RUNG
   // the same network as SCL:
   "m2ConWatOut_TT"(TempIn := "rM2CondWaterOutTemp_C");   // "RTD"
END_REGION

REGION Network 14: M2 Condenser Water In
   RUNG wire#powerrail
      "m2ConWatIn_TT"(TempIn := "rM2CondWaterInTemp_C", Temp_O =>)
   END_RUNG
   // the same network as SCL:
   "m2ConWatIn_TT"(TempIn := "rM2CondWaterInTemp_C");   // "RTD"
END_REGION
END_FUNCTION

FUNCTION "OilTemp" : Void   // FC3, SCL
{ S7_Optimized_Access := 'TRUE' }
VERSION : 0.1
   VAR_TEMP
      m1onoff_temp_real : Real;
      m1OnOff_Enable : Bool;
      m2onoff_temp_real : Real;
      m2OnOff_Enable : Bool;
   END_VAR
BEGIN
   //machine 1 oil on-off temp control 

   #m1onoff_temp_real := "HMI".rM1OilTempSet - "HMI".rM1OilTempHis;
   IF #m1OnOff_Enable AND "m1Oil_TT".Temp_O <= #m1onoff_temp_real AND "HMI".rM1OilTempSet >= "m1Oil_TT".Temp_O THEN
       "AuxOutput".m1OilTempSelenoid := TRUE;
   ELSE
       "AuxOutput".m1OilTempSelenoid := FALSE;
   END_IF;

   //machine 2 oil on-off temp control 

   #m2onoff_temp_real := "HMI".rM2OilTempSet - "HMI".rM2OilTempHis;
   IF #m2OnOff_Enable AND "m2Oil_TT".Temp_O <= #m2onoff_temp_real AND "HMI".rM2OilTempSet >= "m2Oil_TT".Temp_O THEN
       "AuxOutput".m2OilTempSelenoid := TRUE;
   ELSE
       "AuxOutput".m2OilTempSelenoid := FALSE;
   END_IF;
END_FUNCTION

FUNCTION "Out_FC" : Void   // FC4, LAD
{ S7_Optimized_Access := 'TRUE' }
VERSION : 0.1
BEGIN

REGION Network 1: m1 Oil colling line 5 number equipment number 5- 25 valve
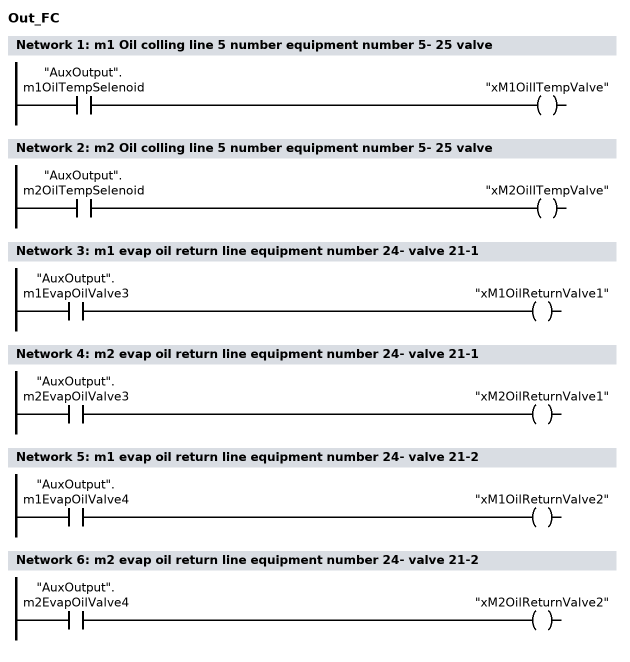
   RUNG wire#powerrail
      Contact( "AuxOutput".m1OilTempSelenoid )
      Coil( "xM1OilITempValve" )
   END_RUNG
   // the same network as SCL:
   "xM1OilITempValve" := "AuxOutput".m1OilTempSelenoid;
END_REGION

REGION Network 2: m2 Oil colling line 5 number equipment number 5- 25 valve
   RUNG wire#powerrail
      Contact( "AuxOutput".m2OilTempSelenoid )
      Coil( "xM2OilITempValve" )
   END_RUNG
   // the same network as SCL:
   "xM2OilITempValve" := "AuxOutput".m2OilTempSelenoid;
END_REGION

REGION Network 3: m1 evap oil return line equipment number 24- valve 21-1
   RUNG wire#powerrail
      Contact( "AuxOutput".m1EvapOilValve3 )
      Coil( "xM1OilReturnValve1" )
   END_RUNG
   // the same network as SCL:
   "xM1OilReturnValve1" := "AuxOutput".m1EvapOilValve3;
END_REGION

REGION Network 4: m2 evap oil return line equipment number 24- valve 21-1
   RUNG wire#powerrail
      Contact( "AuxOutput".m2EvapOilValve3 )
      Coil( "xM2OilReturnValve1" )
   END_RUNG
   // the same network as SCL:
   "xM2OilReturnValve1" := "AuxOutput".m2EvapOilValve3;
END_REGION

REGION Network 5: m1 evap oil return line equipment number 24- valve 21-2
   RUNG wire#powerrail
      Contact( "AuxOutput".m1EvapOilValve4 )
      Coil( "xM1OilReturnValve2" )
   END_RUNG
   // the same network as SCL:
   "xM1OilReturnValve2" := "AuxOutput".m1EvapOilValve4;
END_REGION

REGION Network 6: m2 evap oil return line equipment number 24- valve 21-2
   RUNG wire#powerrail
      Contact( "AuxOutput".m2EvapOilValve4 )
      Coil( "xM2OilReturnValve2" )
   END_RUNG
   // the same network as SCL:
   "xM2OilReturnValve2" := "AuxOutput".m2EvapOilValve4;
END_REGION
END_FUNCTION

FUNCTION "EvapOilLevelControl" : Void   // FC5, LAD
{ S7_Optimized_Access := 'TRUE' }
VERSION : 0.1
   VAR_TEMP
      m1OilLevel1Enable : Bool;
      m1OilDisRunning : Bool;
      m2OilLevel1Enable : Bool;
      m2OilDisRunning : Bool;
   END_VAR
BEGIN

REGION Network 1: M1 Evaparatör oil discharge valfs running
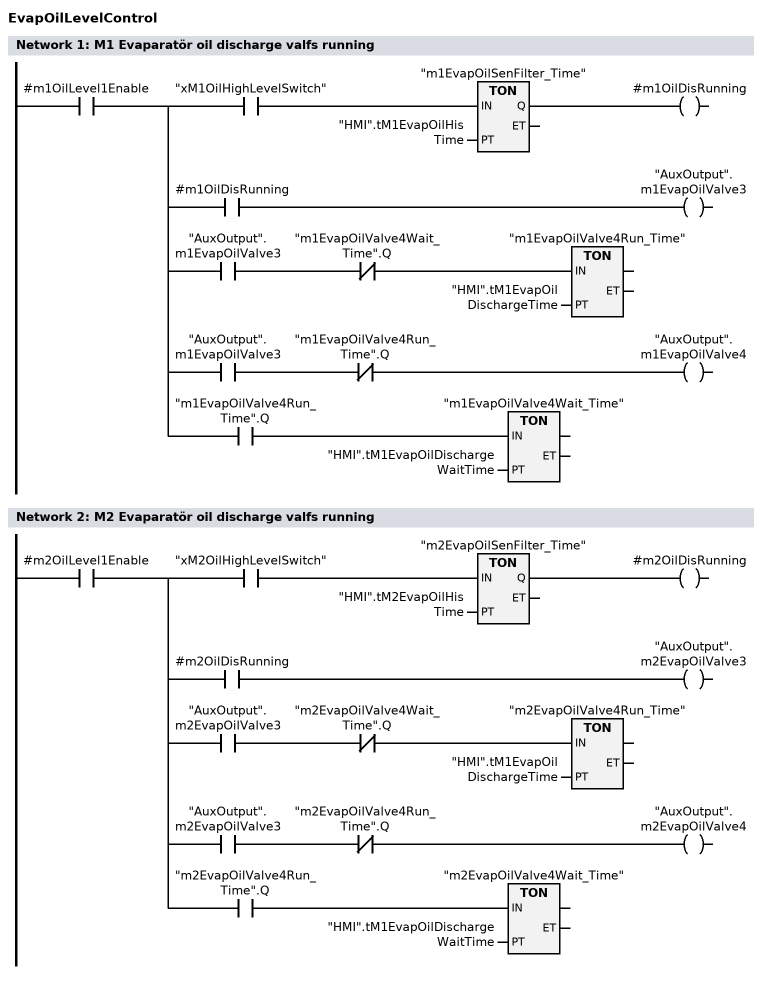
   "m1EvapOilSenFilter_Time".TON(IN := #m1OilLevel1Enable AND "xM1OilHighLevelSwitch",
                           PT := "HMI".tM1EvapOilHisTime);
   #m1OilDisRunning := "m1EvapOilSenFilter_Time".Q;
   "AuxOutput".m1EvapOilValve3 := #m1OilLevel1Enable AND #m1OilDisRunning;
   "m1EvapOilValve4Run_Time".TON(IN := #m1OilLevel1Enable AND "AuxOutput".m1EvapOilValve3 AND NOT "m1EvapOilValve4Wait_Time".Q,
                           PT := "HMI".tM1EvapOilDischargeTime);
   "AuxOutput".m1EvapOilValve4 := #m1OilLevel1Enable AND "AuxOutput".m1EvapOilValve3 AND NOT "m1EvapOilValve4Run_Time".Q;
   "m1EvapOilValve4Wait_Time".TON(IN := #m1OilLevel1Enable AND "m1EvapOilValve4Run_Time".Q,
                           PT := "HMI".tM1EvapOilDischargeWaitTime);
END_REGION

REGION Network 2: M2 Evaparatör oil discharge valfs running
   "m2EvapOilSenFilter_Time".TON(IN := #m2OilLevel1Enable AND "xM2OilHighLevelSwitch",
                           PT := "HMI".tM2EvapOilHisTime);
   #m2OilDisRunning := "m2EvapOilSenFilter_Time".Q;
   "AuxOutput".m2EvapOilValve3 := #m2OilLevel1Enable AND #m2OilDisRunning;
   "m2EvapOilValve4Run_Time".TON(IN := #m2OilLevel1Enable AND "AuxOutput".m2EvapOilValve3 AND NOT "m2EvapOilValve4Wait_Time".Q,
                           PT := "HMI".tM1EvapOilDischargeTime);
   "AuxOutput".m2EvapOilValve4 := #m2OilLevel1Enable AND "AuxOutput".m2EvapOilValve3 AND NOT "m2EvapOilValve4Run_Time".Q;
   "m2EvapOilValve4Wait_Time".TON(IN := #m2OilLevel1Enable AND "m2EvapOilValve4Run_Time".Q,
                           PT := "HMI".tM1EvapOilDischargeWaitTime);
END_REGION
END_FUNCTION

FUNCTION "Alarm" : Void   // FC6, LAD
{ S7_Optimized_Access := 'TRUE' }
VERSION : 0.1
BEGIN

REGION Network 1: M1 Discharge High Pressure Alarm in Dijital Signal
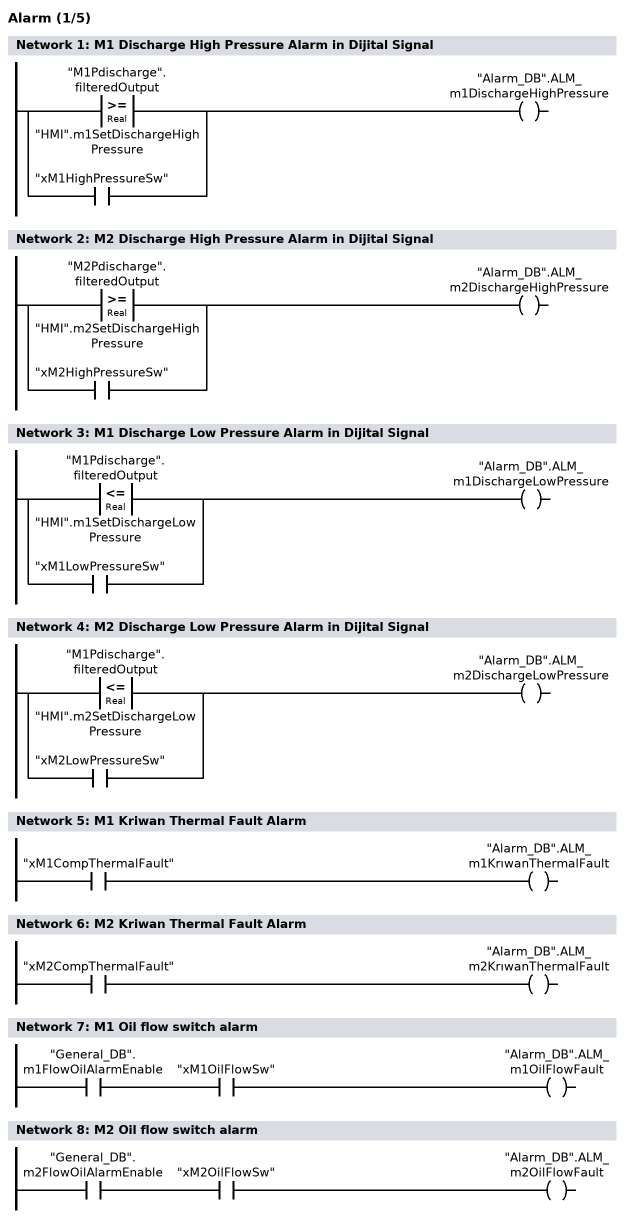
   RUNG wire#powerrail
      { S7_Templates := "SrcType := Real" } GE_Contact(in1 := "M1Pdischarge".filteredOutput, in2 := "HMI".m1SetDischargeHighPressure)
      wire#w1
      Coil( "Alarm_DB".ALM_m1DischargeHighPressure )
   END_RUNG
   RUNG wire#powerrail
      Contact( "xM1HighPressureSw" )
   END_RUNG wire#w1
   // the same network as SCL:
   "Alarm_DB".ALM_m1DischargeHighPressure := ("M1Pdischarge".filteredOutput >= "HMI".m1SetDischargeHighPressure) OR "xM1HighPressureSw";
END_REGION

REGION Network 2: M2 Discharge High Pressure Alarm in Dijital Signal
   RUNG wire#powerrail
      { S7_Templates := "SrcType := Real" } GE_Contact(in1 := "M2Pdischarge".filteredOutput, in2 := "HMI".m2SetDischargeHighPressure)
      wire#w1
      Coil( "Alarm_DB".ALM_m2DischargeHighPressure )
   END_RUNG
   RUNG wire#powerrail
      Contact( "xM2HighPressureSw" )
   END_RUNG wire#w1
   // the same network as SCL:
   "Alarm_DB".ALM_m2DischargeHighPressure := ("M2Pdischarge".filteredOutput >= "HMI".m2SetDischargeHighPressure) OR "xM2HighPressureSw";
END_REGION

REGION Network 3: M1 Discharge Low Pressure Alarm in Dijital Signal
   RUNG wire#powerrail
      { S7_Templates := "SrcType := Real" } LE_Contact(in1 := "M1Pdischarge".filteredOutput, in2 := "HMI".m1SetDischargeLowPressure)
      wire#w1
      Coil( "Alarm_DB".ALM_m1DischargeLowPressure )
   END_RUNG
   RUNG wire#powerrail
      Contact( "xM1LowPressureSw" )
   END_RUNG wire#w1
   // the same network as SCL:
   "Alarm_DB".ALM_m1DischargeLowPressure := ("M1Pdischarge".filteredOutput <= "HMI".m1SetDischargeLowPressure) OR "xM1LowPressureSw";
END_REGION

REGION Network 4: M2 Discharge Low Pressure Alarm in Dijital Signal
   RUNG wire#powerrail
      { S7_Templates := "SrcType := Real" } LE_Contact(in1 := "M1Pdischarge".filteredOutput, in2 := "HMI".m2SetDischargeLowPressure)
      wire#w1
      Coil( "Alarm_DB".ALM_m2DischargeLowPressure )
   END_RUNG
   RUNG wire#powerrail
      Contact( "xM2LowPressureSw" )
   END_RUNG wire#w1
   // the same network as SCL:
   "Alarm_DB".ALM_m2DischargeLowPressure := ("M1Pdischarge".filteredOutput <= "HMI".m2SetDischargeLowPressure) OR "xM2LowPressureSw";
END_REGION

REGION Network 5: M1 Kriwan Thermal Fault Alarm
   RUNG wire#powerrail
      Contact( "xM1CompThermalFault" )
      Coil( "Alarm_DB".ALM_m1KrıwanThermalFault )
   END_RUNG
   // the same network as SCL:
   "Alarm_DB".ALM_m1KrıwanThermalFault := "xM1CompThermalFault";
END_REGION

REGION Network 6: M2 Kriwan Thermal Fault Alarm
   RUNG wire#powerrail
      Contact( "xM2CompThermalFault" )
      Coil( "Alarm_DB".ALM_m2KrıwanThermalFault )
   END_RUNG
   // the same network as SCL:
   "Alarm_DB".ALM_m2KrıwanThermalFault := "xM2CompThermalFault";
END_REGION

REGION Network 7: M1 Oil flow switch alarm
   RUNG wire#powerrail
      Contact( "General_DB".m1FlowOilAlarmEnable )
      Contact( "xM1OilFlowSw" )
      Coil( "Alarm_DB".ALM_m1OilFlowFault )
   END_RUNG
   // the same network as SCL:
   "Alarm_DB".ALM_m1OilFlowFault := "General_DB".m1FlowOilAlarmEnable AND "xM1OilFlowSw";
END_REGION

REGION Network 8: M2 Oil flow switch alarm
   RUNG wire#powerrail
      Contact( "General_DB".m2FlowOilAlarmEnable )
      Contact( "xM2OilFlowSw" )
      Coil( "Alarm_DB".ALM_m2OilFlowFault )
   END_RUNG
   // the same network as SCL:
   "Alarm_DB".ALM_m2OilFlowFault := "General_DB".m2FlowOilAlarmEnable AND "xM2OilFlowSw";
END_REGION

REGION Network 9: M1 Condens flow switch alarm stop
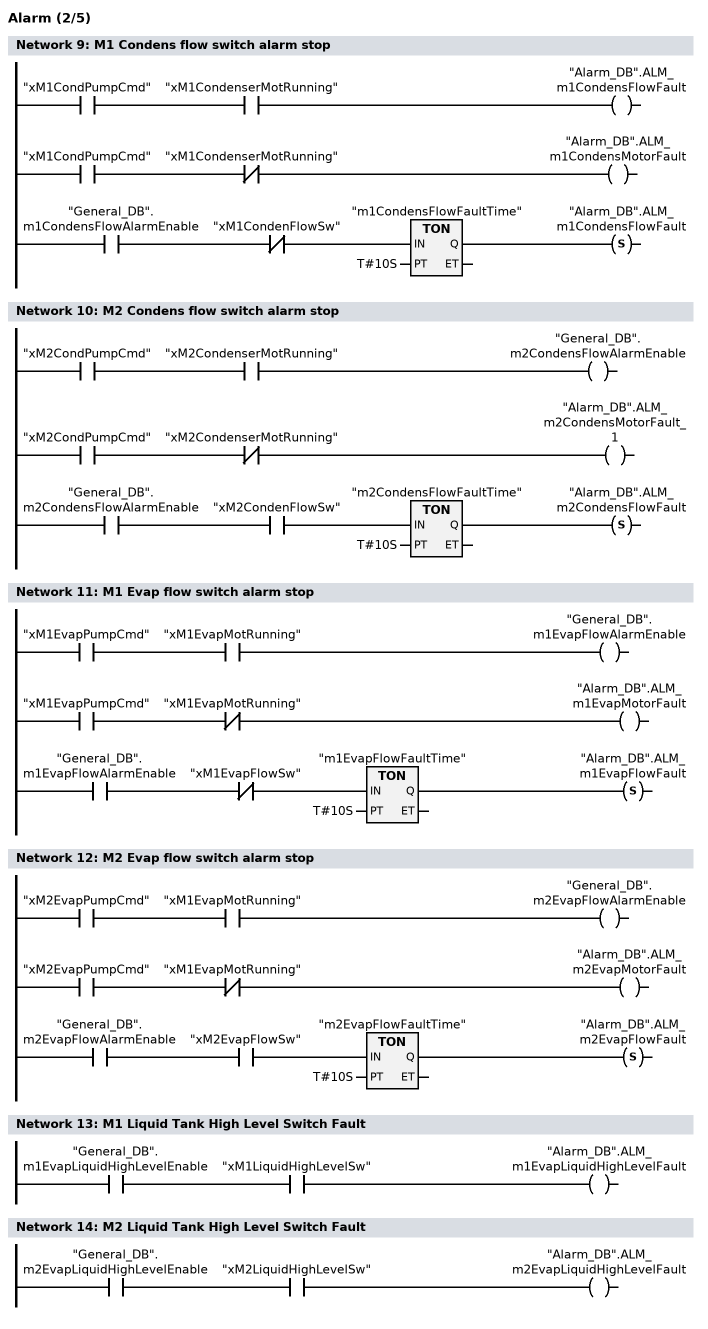
   "Alarm_DB".ALM_m1CondensFlowFault := "xM1CondPumpCmd" AND "xM1CondenserMotRunning";
   "Alarm_DB".ALM_m1CondensMotorFault := "xM1CondPumpCmd" AND NOT "xM1CondenserMotRunning";
   "m1CondensFlowFaultTime".TON(IN := "General_DB".m1CondensFlowAlarmEnable AND NOT "xM1CondenFlowSw",
                           PT := T#10S);
   IF "m1CondensFlowFaultTime".Q THEN "Alarm_DB".ALM_m1CondensFlowFault := TRUE; END_IF;
END_REGION

REGION Network 10: M2 Condens flow switch alarm stop
   "General_DB".m2CondensFlowAlarmEnable := "xM2CondPumpCmd" AND "xM2CondenserMotRunning";
   "Alarm_DB".ALM_m2CondensMotorFault_1 := "xM2CondPumpCmd" AND NOT "xM2CondenserMotRunning";
   "m2CondensFlowFaultTime".TON(IN := "General_DB".m2CondensFlowAlarmEnable AND "xM2CondenFlowSw", PT := T#10S);
   IF "m2CondensFlowFaultTime".Q THEN "Alarm_DB".ALM_m2CondensFlowFault := TRUE; END_IF;
END_REGION

REGION Network 11: M1 Evap flow switch alarm stop
   "General_DB".m1EvapFlowAlarmEnable := "xM1EvapPumpCmd" AND "xM1EvapMotRunning";
   "Alarm_DB".ALM_m1EvapMotorFault := "xM1EvapPumpCmd" AND NOT "xM1EvapMotRunning";
   "m1EvapFlowFaultTime".TON(IN := "General_DB".m1EvapFlowAlarmEnable AND NOT "xM1EvapFlowSw", PT := T#10S);
   IF "m1EvapFlowFaultTime".Q THEN "Alarm_DB".ALM_m1EvapFlowFault := TRUE; END_IF;
END_REGION

REGION Network 12: M2 Evap flow switch alarm stop
   "General_DB".m2EvapFlowAlarmEnable := "xM2EvapPumpCmd" AND "xM1EvapMotRunning";
   "Alarm_DB".ALM_m2EvapMotorFault := "xM2EvapPumpCmd" AND NOT "xM1EvapMotRunning";
   "m2EvapFlowFaultTime".TON(IN := "General_DB".m2EvapFlowAlarmEnable AND "xM2EvapFlowSw", PT := T#10S);
   IF "m2EvapFlowFaultTime".Q THEN "Alarm_DB".ALM_m2EvapFlowFault := TRUE; END_IF;
END_REGION

REGION Network 13: M1 Liquid Tank High Level Switch Fault
   RUNG wire#powerrail
      Contact( "General_DB".m1EvapLiquidHighLevelEnable )
      Contact( "xM1LiquidHighLevelSw" )
      Coil( "Alarm_DB".ALM_m1EvapLiquidHighLevelFault )
   END_RUNG
   // the same network as SCL:
   "Alarm_DB".ALM_m1EvapLiquidHighLevelFault := "General_DB".m1EvapLiquidHighLevelEnable AND "xM1LiquidHighLevelSw";
END_REGION

REGION Network 14: M2 Liquid Tank High Level Switch Fault
   RUNG wire#powerrail
      Contact( "General_DB".m2EvapLiquidHighLevelEnable )
      Contact( "xM2LiquidHighLevelSw" )
      Coil( "Alarm_DB".ALM_m2EvapLiquidHighLevelFault )
   END_RUNG
   // the same network as SCL:
   "Alarm_DB".ALM_m2EvapLiquidHighLevelFault := "General_DB".m2EvapLiquidHighLevelEnable AND "xM2LiquidHighLevelSw";
END_REGION

REGION Network 15: M1 Liquid Tank Low Level Switch Fault
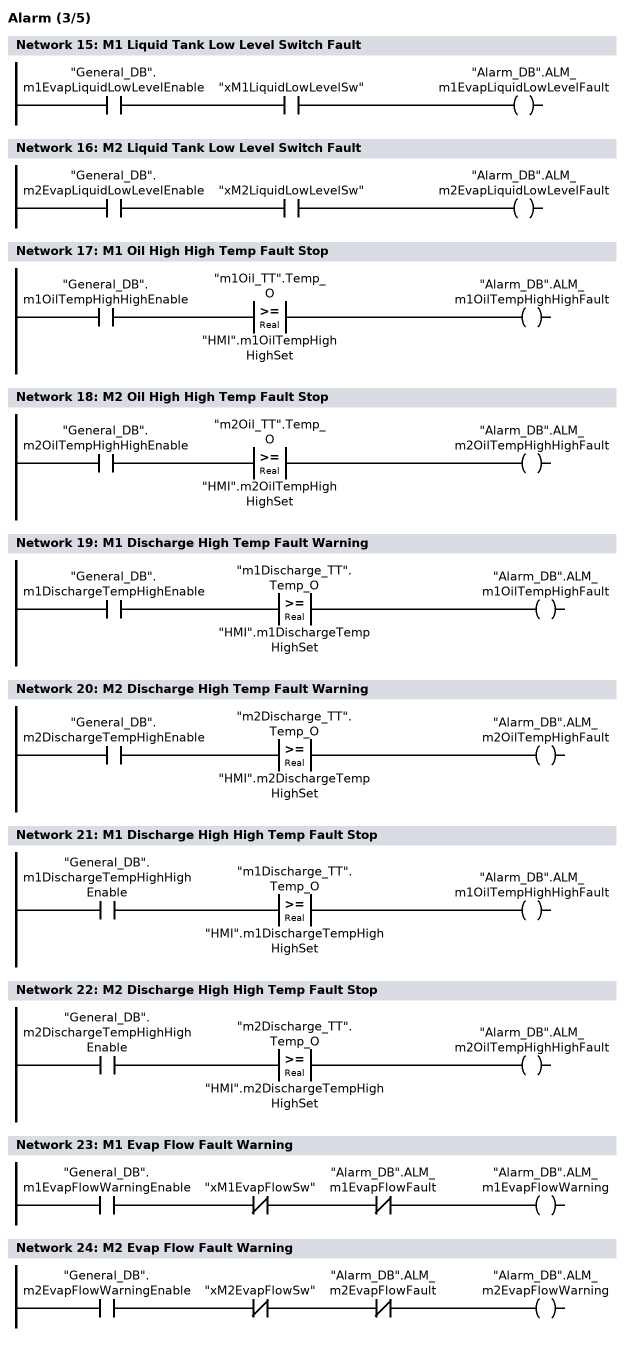
   RUNG wire#powerrail
      Contact( "General_DB".m1EvapLiquidLowLevelEnable )
      Contact( "xM1LiquidLowLevelSw" )
      Coil( "Alarm_DB".ALM_m1EvapLiquidLowLevelFault )
   END_RUNG
   // the same network as SCL:
   "Alarm_DB".ALM_m1EvapLiquidLowLevelFault := "General_DB".m1EvapLiquidLowLevelEnable AND "xM1LiquidLowLevelSw";
END_REGION

REGION Network 16: M2 Liquid Tank Low Level Switch Fault
   RUNG wire#powerrail
      Contact( "General_DB".m2EvapLiquidLowLevelEnable )
      Contact( "xM2LiquidLowLevelSw" )
      Coil( "Alarm_DB".ALM_m2EvapLiquidLowLevelFault )
   END_RUNG
   // the same network as SCL:
   "Alarm_DB".ALM_m2EvapLiquidLowLevelFault := "General_DB".m2EvapLiquidLowLevelEnable AND "xM2LiquidLowLevelSw";
END_REGION

REGION Network 17: M1 Oil High High Temp Fault Stop
   RUNG wire#powerrail
      Contact( "General_DB".m1OilTempHighHighEnable )
      { S7_Templates := "SrcType := Real" } GE_Contact(in1 := "m1Oil_TT".Temp_O, in2 := "HMI".m1OilTempHighHighSet)
      Coil( "Alarm_DB".ALM_m1OilTempHighHighFault )
   END_RUNG
   // the same network as SCL:
   "Alarm_DB".ALM_m1OilTempHighHighFault := "General_DB".m1OilTempHighHighEnable AND ("m1Oil_TT".Temp_O >= "HMI".m1OilTempHighHighSet);
END_REGION

REGION Network 18: M2 Oil High High Temp Fault Stop
   RUNG wire#powerrail
      Contact( "General_DB".m2OilTempHighHighEnable )
      { S7_Templates := "SrcType := Real" } GE_Contact(in1 := "m2Oil_TT".Temp_O, in2 := "HMI".m2OilTempHighHighSet)
      Coil( "Alarm_DB".ALM_m2OilTempHighHighFault )
   END_RUNG
   // the same network as SCL:
   "Alarm_DB".ALM_m2OilTempHighHighFault := "General_DB".m2OilTempHighHighEnable AND ("m2Oil_TT".Temp_O >= "HMI".m2OilTempHighHighSet);
END_REGION

REGION Network 19: M1 Discharge High Temp Fault Warning
   RUNG wire#powerrail
      Contact( "General_DB".m1DischargeTempHighEnable )
      { S7_Templates := "SrcType := Real" } GE_Contact(in1 := "m1Discharge_TT".Temp_O, in2 := "HMI".m1DischargeTempHighSet)
      Coil( "Alarm_DB".ALM_m1OilTempHighFault )
   END_RUNG
   // the same network as SCL:
   "Alarm_DB".ALM_m1OilTempHighFault := "General_DB".m1DischargeTempHighEnable AND ("m1Discharge_TT".Temp_O >= "HMI".m1DischargeTempHighSet);
END_REGION

REGION Network 20: M2 Discharge High Temp Fault Warning
   RUNG wire#powerrail
      Contact( "General_DB".m2DischargeTempHighEnable )
      { S7_Templates := "SrcType := Real" } GE_Contact(in1 := "m2Discharge_TT".Temp_O, in2 := "HMI".m2DischargeTempHighSet)
      Coil( "Alarm_DB".ALM_m2OilTempHighFault )
   END_RUNG
   // the same network as SCL:
   "Alarm_DB".ALM_m2OilTempHighFault := "General_DB".m2DischargeTempHighEnable AND ("m2Discharge_TT".Temp_O >= "HMI".m2DischargeTempHighSet);
END_REGION

REGION Network 21: M1 Discharge High High Temp Fault Stop
   RUNG wire#powerrail
      Contact( "General_DB".m1DischargeTempHighHighEnable )
      { S7_Templates := "SrcType := Real" } GE_Contact(in1 := "m1Discharge_TT".Temp_O, in2 := "HMI".m1DischargeTempHighHighSet)
      Coil( "Alarm_DB".ALM_m1OilTempHighHighFault )
   END_RUNG
   // the same network as SCL:
   "Alarm_DB".ALM_m1OilTempHighHighFault := "General_DB".m1DischargeTempHighHighEnable AND ("m1Discharge_TT".Temp_O >= "HMI".m1DischargeTempHighHighSet);
END_REGION

REGION Network 22: M2 Discharge High High Temp Fault Stop
   RUNG wire#powerrail
      Contact( "General_DB".m2DischargeTempHighHighEnable )
      { S7_Templates := "SrcType := Real" } GE_Contact(in1 := "m2Discharge_TT".Temp_O, in2 := "HMI".m2DischargeTempHighHighSet)
      Coil( "Alarm_DB".ALM_m2OilTempHighHighFault )
   END_RUNG
   // the same network as SCL:
   "Alarm_DB".ALM_m2OilTempHighHighFault := "General_DB".m2DischargeTempHighHighEnable AND ("m2Discharge_TT".Temp_O >= "HMI".m2DischargeTempHighHighSet);
END_REGION

REGION Network 23: M1 Evap Flow Fault Warning
   RUNG wire#powerrail
      Contact( "General_DB".m1EvapFlowWarningEnable )
      I_Contact( "xM1EvapFlowSw" )
      I_Contact( "Alarm_DB".ALM_m1EvapFlowFault )
      Coil( "Alarm_DB".ALM_m1EvapFlowWarning )
   END_RUNG
   // the same network as SCL:
   "Alarm_DB".ALM_m1EvapFlowWarning := "General_DB".m1EvapFlowWarningEnable AND NOT "xM1EvapFlowSw" AND NOT "Alarm_DB".ALM_m1EvapFlowFault;
END_REGION

REGION Network 24: M2 Evap Flow Fault Warning
   RUNG wire#powerrail
      Contact( "General_DB".m2EvapFlowWarningEnable )
      I_Contact( "xM2EvapFlowSw" )
      I_Contact( "Alarm_DB".ALM_m2EvapFlowFault )
      Coil( "Alarm_DB".ALM_m2EvapFlowWarning )
   END_RUNG
   // the same network as SCL:
   "Alarm_DB".ALM_m2EvapFlowWarning := "General_DB".m2EvapFlowWarningEnable AND NOT "xM2EvapFlowSw" AND NOT "Alarm_DB".ALM_m2EvapFlowFault;
END_REGION

REGION Network 25: M1 Condens Flow Fault Warning
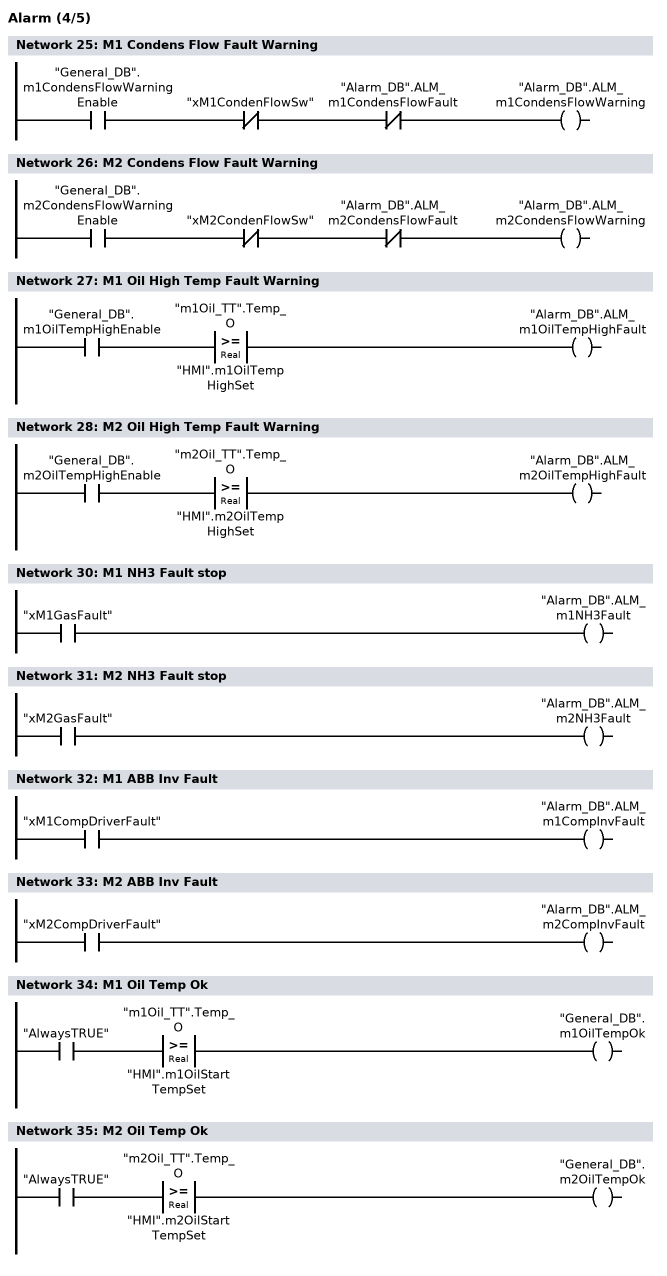
   RUNG wire#powerrail
      Contact( "General_DB".m1CondensFlowWarningEnable )
      I_Contact( "xM1CondenFlowSw" )
      I_Contact( "Alarm_DB".ALM_m1CondensFlowFault )
      Coil( "Alarm_DB".ALM_m1CondensFlowWarning )
   END_RUNG
   // the same network as SCL:
   "Alarm_DB".ALM_m1CondensFlowWarning := "General_DB".m1CondensFlowWarningEnable AND NOT "xM1CondenFlowSw" AND NOT "Alarm_DB".ALM_m1CondensFlowFault;
END_REGION

REGION Network 26: M2 Condens Flow Fault Warning
   RUNG wire#powerrail
      Contact( "General_DB".m2CondensFlowWarningEnable )
      I_Contact( "xM2CondenFlowSw" )
      I_Contact( "Alarm_DB".ALM_m2CondensFlowFault )
      Coil( "Alarm_DB".ALM_m2CondensFlowWarning )
   END_RUNG
   // the same network as SCL:
   "Alarm_DB".ALM_m2CondensFlowWarning := "General_DB".m2CondensFlowWarningEnable AND NOT "xM2CondenFlowSw" AND NOT "Alarm_DB".ALM_m2CondensFlowFault;
END_REGION

REGION Network 27: M1 Oil High Temp Fault Warning
   RUNG wire#powerrail
      Contact( "General_DB".m1OilTempHighEnable )
      { S7_Templates := "SrcType := Real" } GE_Contact(in1 := "m1Oil_TT".Temp_O, in2 := "HMI".m1OilTempHighSet)
      Coil( "Alarm_DB".ALM_m1OilTempHighFault )
   END_RUNG
   // the same network as SCL:
   "Alarm_DB".ALM_m1OilTempHighFault := "General_DB".m1OilTempHighEnable AND ("m1Oil_TT".Temp_O >= "HMI".m1OilTempHighSet);
END_REGION

REGION Network 28: M2 Oil High Temp Fault Warning
   RUNG wire#powerrail
      Contact( "General_DB".m2OilTempHighEnable )
      { S7_Templates := "SrcType := Real" } GE_Contact(in1 := "m2Oil_TT".Temp_O, in2 := "HMI".m2OilTempHighSet)
      Coil( "Alarm_DB".ALM_m2OilTempHighFault )
   END_RUNG
   // the same network as SCL:
   "Alarm_DB".ALM_m2OilTempHighFault := "General_DB".m2OilTempHighEnable AND ("m2Oil_TT".Temp_O >= "HMI".m2OilTempHighSet);
END_REGION

REGION Network 29: IF Level nahe Grenze → WARNUNG (Bu sorulacak ona göre yazılacak)
END_REGION

REGION Network 30: M1 NH3 Fault stop
   RUNG wire#powerrail
      Contact( "xM1GasFault" )
      Coil( "Alarm_DB".ALM_m1NH3Fault )
   END_RUNG
   // the same network as SCL:
   "Alarm_DB".ALM_m1NH3Fault := "xM1GasFault";
END_REGION

REGION Network 31: M2 NH3 Fault stop
   RUNG wire#powerrail
      Contact( "xM2GasFault" )
      Coil( "Alarm_DB".ALM_m2NH3Fault )
   END_RUNG
   // the same network as SCL:
   "Alarm_DB".ALM_m2NH3Fault := "xM2GasFault";
END_REGION

REGION Network 32: M1 ABB Inv Fault
   RUNG wire#powerrail
      Contact( "xM1CompDriverFault" )
      Coil( "Alarm_DB".ALM_m1CompInvFault )
   END_RUNG
   // the same network as SCL:
   "Alarm_DB".ALM_m1CompInvFault := "xM1CompDriverFault";
END_REGION

REGION Network 33: M2 ABB Inv Fault
   RUNG wire#powerrail
      Contact( "xM2CompDriverFault" )
      Coil( "Alarm_DB".ALM_m2CompInvFault )
   END_RUNG
   // the same network as SCL:
   "Alarm_DB".ALM_m2CompInvFault := "xM2CompDriverFault";
END_REGION

REGION Network 34: M1 Oil Temp Ok
   RUNG wire#powerrail
      Contact( "AlwaysTRUE" )
      { S7_Templates := "SrcType := Real" } GE_Contact(in1 := "m1Oil_TT".Temp_O, in2 := "HMI".m1OilStartTempSet)
      Coil( "General_DB".m1OilTempOk )
   END_RUNG
   // the same network as SCL:
   "General_DB".m1OilTempOk := "AlwaysTRUE" AND ("m1Oil_TT".Temp_O >= "HMI".m1OilStartTempSet);
END_REGION

REGION Network 35: M2 Oil Temp Ok
   RUNG wire#powerrail
      Contact( "AlwaysTRUE" )
      { S7_Templates := "SrcType := Real" } GE_Contact(in1 := "m2Oil_TT".Temp_O, in2 := "HMI".m2OilStartTempSet)
      Coil( "General_DB".m2OilTempOk )
   END_RUNG
   // the same network as SCL:
   "General_DB".m2OilTempOk := "AlwaysTRUE" AND ("m2Oil_TT".Temp_O >= "HMI".m2OilStartTempSet);
END_REGION

REGION Network 36: Phase Protection relay fault
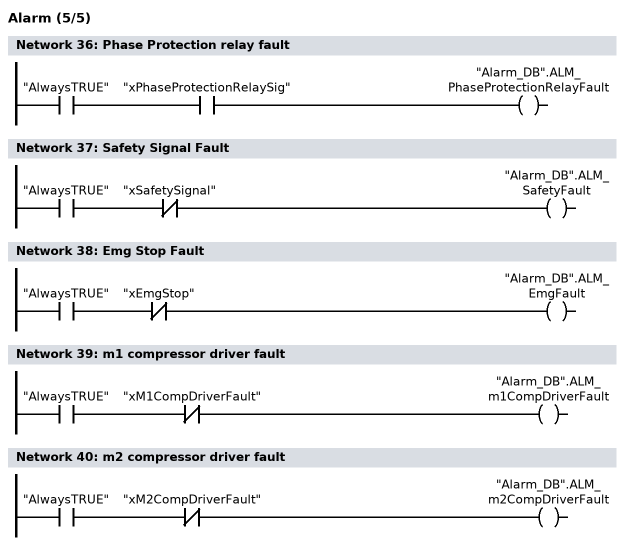
   RUNG wire#powerrail
      Contact( "AlwaysTRUE" )
      Contact( "xPhaseProtectionRelaySig" )
      Coil( "Alarm_DB".ALM_PhaseProtectionRelayFault )
   END_RUNG
   // the same network as SCL:
   "Alarm_DB".ALM_PhaseProtectionRelayFault := "AlwaysTRUE" AND "xPhaseProtectionRelaySig";
END_REGION

REGION Network 37: Safety Signal Fault
   RUNG wire#powerrail
      Contact( "AlwaysTRUE" )
      I_Contact( "xSafetySignal" )
      Coil( "Alarm_DB".ALM_SafetyFault )
   END_RUNG
   // the same network as SCL:
   "Alarm_DB".ALM_SafetyFault := "AlwaysTRUE" AND NOT "xSafetySignal";
END_REGION

REGION Network 38: Emg Stop Fault
   RUNG wire#powerrail
      Contact( "AlwaysTRUE" )
      I_Contact( "xEmgStop" )
      Coil( "Alarm_DB".ALM_EmgFault )
   END_RUNG
   // the same network as SCL:
   "Alarm_DB".ALM_EmgFault := "AlwaysTRUE" AND NOT "xEmgStop";
END_REGION

REGION Network 39: m1 compressor driver fault
   RUNG wire#powerrail
      Contact( "AlwaysTRUE" )
      I_Contact( "xM1CompDriverFault" )
      Coil( "Alarm_DB".ALM_m1CompDriverFault )
   END_RUNG
   // the same network as SCL:
   "Alarm_DB".ALM_m1CompDriverFault := "AlwaysTRUE" AND NOT "xM1CompDriverFault";
END_REGION

REGION Network 40: m2 compressor driver fault
   RUNG wire#powerrail
      Contact( "AlwaysTRUE" )
      I_Contact( "xM2CompDriverFault" )
      Coil( "Alarm_DB".ALM_m2CompDriverFault )
   END_RUNG
   // the same network as SCL:
   "Alarm_DB".ALM_m2CompDriverFault := "AlwaysTRUE" AND NOT "xM2CompDriverFault";
END_REGION
END_FUNCTION

FUNCTION "Machine1_Start" : Void   // FC7, LAD
{ S7_Optimized_Access := 'TRUE' }
VERSION : 0.1
   VAR_TEMP
      Machine1_Ready : Bool;
      clock_yrd1 : Bool;
      clock_yrd2 : Bool;
      clock_yrd3 : Bool;
   END_VAR
   VAR_TEMP   // added for the SCL form of the ladder/FBD networks
      _w1 : Bool;
      _w2 : Bool;
   END_VAR
BEGIN

REGION Network 1: Machine 1 ready conditions
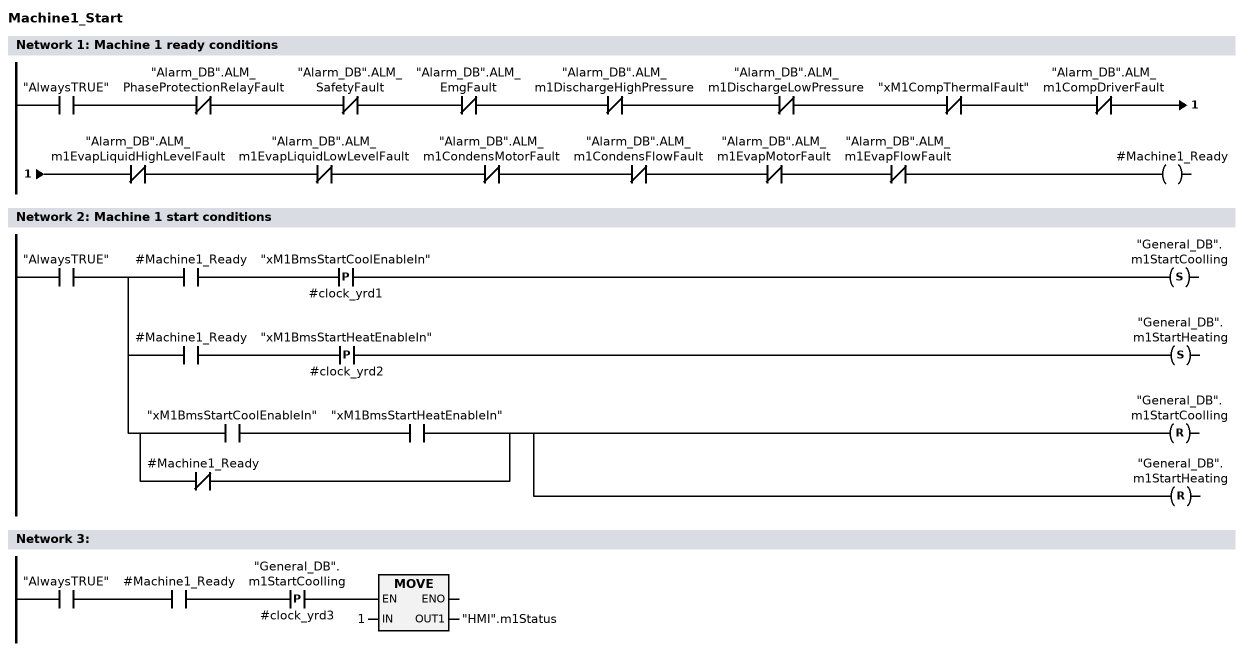
   RUNG wire#powerrail
      Contact( "AlwaysTRUE" )
      I_Contact( "Alarm_DB".ALM_PhaseProtectionRelayFault )
      I_Contact( "Alarm_DB".ALM_SafetyFault )
      I_Contact( "Alarm_DB".ALM_EmgFault )
      I_Contact( "Alarm_DB".ALM_m1DischargeHighPressure )
      I_Contact( "Alarm_DB".ALM_m1DischargeLowPressure )
      I_Contact( "xM1CompThermalFault" )
      I_Contact( "Alarm_DB".ALM_m1CompDriverFault )
      I_Contact( "Alarm_DB".ALM_m1EvapLiquidHighLevelFault )
      I_Contact( "Alarm_DB".ALM_m1EvapLiquidLowLevelFault )
      I_Contact( "Alarm_DB".ALM_m1CondensMotorFault )
      I_Contact( "Alarm_DB".ALM_m1CondensFlowFault )
      I_Contact( "Alarm_DB".ALM_m1EvapMotorFault )
      I_Contact( "Alarm_DB".ALM_m1EvapFlowFault )
      Coil( #Machine1_Ready )
   END_RUNG
   // the same network as SCL:
   #Machine1_Ready := "AlwaysTRUE" AND NOT "Alarm_DB".ALM_PhaseProtectionRelayFault AND NOT "Alarm_DB".ALM_SafetyFault AND NOT "Alarm_DB".ALM_EmgFault AND NOT "Alarm_DB".ALM_m1DischargeHighPressure AND NOT "Alarm_DB".ALM_m1DischargeLowPressure AND NOT "xM1CompThermalFault" AND NOT "Alarm_DB".ALM_m1CompDriverFault AND NOT "Alarm_DB".ALM_m1EvapLiquidHighLevelFault AND NOT "Alarm_DB".ALM_m1EvapLiquidLowLevelFault AND NOT "Alarm_DB".ALM_m1CondensMotorFault AND NOT "Alarm_DB".ALM_m1CondensFlowFault AND NOT "Alarm_DB".ALM_m1EvapMotorFault AND NOT "Alarm_DB".ALM_m1EvapFlowFault;
END_REGION

REGION Network 2: Machine 1 start conditions
   RUNG wire#powerrail
      Contact( "AlwaysTRUE" )
      wire#w1
      Contact( #Machine1_Ready )
      P_Contact(operand := "xM1BmsStartCoolEnableIn", bit := #clock_yrd1)
      S_Coil( "General_DB".m1StartCoolling )
   END_RUNG
   RUNG wire#w1
      Contact( #Machine1_Ready )
      P_Contact(operand := "xM1BmsStartHeatEnableIn", bit := #clock_yrd2)
      S_Coil( "General_DB".m1StartHeating )
   END_RUNG
   RUNG wire#w1
      Contact( "xM1BmsStartCoolEnableIn" )
      Contact( "xM1BmsStartHeatEnableIn" )
      wire#w2
      R_Coil( "General_DB".m1StartCoolling )
   END_RUNG
   RUNG wire#w1
      I_Contact( #Machine1_Ready )
   END_RUNG wire#w2
   RUNG wire#w2
      R_Coil( "General_DB".m1StartHeating )
   END_RUNG
   // the same network as SCL:
   #_w1 := "AlwaysTRUE" AND #Machine1_Ready AND "xM1BmsStartCoolEnableIn" AND NOT #clock_yrd1;   // rising edge of "xM1BmsStartCoolEnableIn"
   #clock_yrd1 := "xM1BmsStartCoolEnableIn";
   IF #_w1 THEN "General_DB".m1StartCoolling := TRUE; END_IF;
   #_w2 := "AlwaysTRUE" AND #Machine1_Ready AND "xM1BmsStartHeatEnableIn" AND NOT #clock_yrd2;   // rising edge of "xM1BmsStartHeatEnableIn"
   #clock_yrd2 := "xM1BmsStartHeatEnableIn";
   IF #_w2 THEN "General_DB".m1StartHeating := TRUE; END_IF;
   IF "AlwaysTRUE" AND (("xM1BmsStartCoolEnableIn" AND "xM1BmsStartHeatEnableIn") OR NOT #Machine1_Ready) THEN
       "General_DB".m1StartCoolling := FALSE;
       "General_DB".m1StartHeating := FALSE;
   END_IF;
END_REGION

REGION Network 3
   RUNG wire#powerrail
      Contact( "AlwaysTRUE" )
      Contact( #Machine1_Ready )
      P_Contact(operand := "General_DB".m1StartCoolling, bit := #clock_yrd3)
      Move(in := 1, out1 => "HMI".m1Status)
   END_RUNG
   // the same network as SCL:
   #_w1 := "AlwaysTRUE" AND #Machine1_Ready AND "General_DB".m1StartCoolling AND NOT #clock_yrd3;   // rising edge of "General_DB".m1StartCoolling
   #clock_yrd3 := "General_DB".m1StartCoolling;
   IF #_w1 THEN "HMI".m1Status := 1; END_IF;
END_REGION
END_FUNCTION

FUNCTION "Machine_TempSet" : Void   // FC8, LAD
{ S7_Optimized_Access := 'TRUE' }
VERSION : 0.1
BEGIN

REGION Network 1: m1 Temp set scale
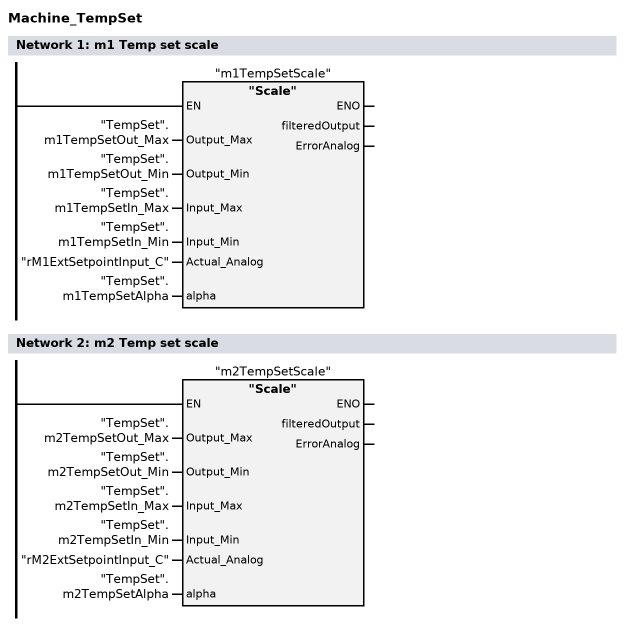
   RUNG wire#powerrail
      "m1TempSetScale"(Output_Max := "TempSet".m1TempSetOut_Max, Output_Min := "TempSet".m1TempSetOut_Min, Input_Max := "TempSet".m1TempSetIn_Max, Input_Min := "TempSet".m1TempSetIn_Min, Actual_Analog := "rM1ExtSetpointInput_C", alpha := "TempSet".m1TempSetAlpha, filteredOutput =>, ErrorAnalog =>)
   END_RUNG
   // the same network as SCL:
   "m1TempSetScale"(Output_Max := "TempSet".m1TempSetOut_Max,   // "Scale"
                    Output_Min := "TempSet".m1TempSetOut_Min,
                    Input_Max := "TempSet".m1TempSetIn_Max,
                    Input_Min := "TempSet".m1TempSetIn_Min,
                    Actual_Analog := "rM1ExtSetpointInput_C",
                    alpha := "TempSet".m1TempSetAlpha);
END_REGION

REGION Network 2: m2 Temp set scale
   RUNG wire#powerrail
      "m2TempSetScale"(Output_Max := "TempSet".m2TempSetOut_Max, Output_Min := "TempSet".m2TempSetOut_Min, Input_Max := "TempSet".m2TempSetIn_Max, Input_Min := "TempSet".m2TempSetIn_Min, Actual_Analog := "rM2ExtSetpointInput_C", alpha := "TempSet".m2TempSetAlpha, filteredOutput =>, ErrorAnalog =>)
   END_RUNG
   // the same network as SCL:
   "m2TempSetScale"(Output_Max := "TempSet".m2TempSetOut_Max,   // "Scale"
                    Output_Min := "TempSet".m2TempSetOut_Min,
                    Input_Max := "TempSet".m2TempSetIn_Max,
                    Input_Min := "TempSet".m2TempSetIn_Min,
                    Actual_Analog := "rM2ExtSetpointInput_C",
                    alpha := "TempSet".m2TempSetAlpha);
END_REGION
END_FUNCTION

ORGANIZATION_BLOCK "Main"   // OB1, LAD, ProgramCycle
TITLE = "Main Program Sweep (Cycle)"
{ S7_Optimized_Access := 'TRUE' }
VERSION : 0.1
   VAR_INPUT
      Initial_Call : Bool;   // Initial call of this OB
      Remanence : Bool;   // =True, if remanent data are available
   END_VAR
BEGIN
END_ORGANIZATION_BLOCK

ORGANIZATION_BLOCK "PID_Control"   // OB30, LAD, CyclicInterrupt
{ S7_Optimized_Access := 'TRUE' }
VERSION : 0.1
   VAR_INPUT
      Initial_Call : Bool;   // Initial call of this OB
      Event_Count : Int;   // Events discarded
   END_VAR
BEGIN

REGION Network 1: machine 1 compressor pid
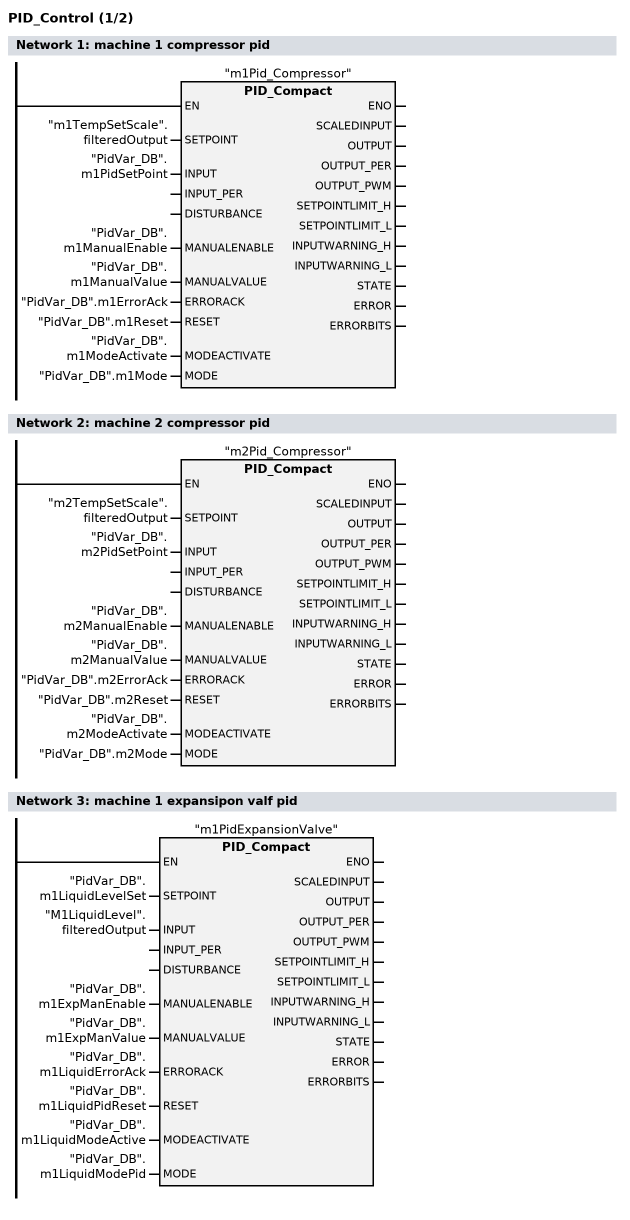
   "m1Pid_Compressor"(Setpoint := "m1TempSetScale".filteredOutput,   // PID_Compact
                      Input := "PidVar_DB".m1PidSetPoint,
                      ManualEnable := "PidVar_DB".m1ManualEnable,
                      ManualValue := "PidVar_DB".m1ManualValue,
                      ErrorAck := "PidVar_DB".m1ErrorAck,
                      Reset := "PidVar_DB".m1Reset,
                      ModeActivate := "PidVar_DB".m1ModeActivate,
                      Mode := "PidVar_DB".m1Mode);
END_REGION

REGION Network 2: machine 2 compressor pid
   "m2Pid_Compressor"(Setpoint := "m2TempSetScale".filteredOutput,   // PID_Compact
                      Input := "PidVar_DB".m2PidSetPoint,
                      ManualEnable := "PidVar_DB".m2ManualEnable,
                      ManualValue := "PidVar_DB".m2ManualValue,
                      ErrorAck := "PidVar_DB".m2ErrorAck,
                      Reset := "PidVar_DB".m2Reset,
                      ModeActivate := "PidVar_DB".m2ModeActivate,
                      Mode := "PidVar_DB".m2Mode);
END_REGION

REGION Network 3: machine 1 expansipon valf pid
   "m1PidExpansionValve"(Setpoint := "PidVar_DB".m1LiquidLevelSet,   // PID_Compact
                         Input := "M1LiquidLevel".filteredOutput,
                         ManualEnable := "PidVar_DB".m1ExpManEnable,
                         ManualValue := "PidVar_DB".m1ExpManValue,
                         ErrorAck := "PidVar_DB".m1LiquidErrorAck,
                         Reset := "PidVar_DB".m1LiquidPidReset,
                         ModeActivate := "PidVar_DB".m1LiquidModeActive,
                         Mode := "PidVar_DB".m1LiquidModePid);
END_REGION

REGION Network 4: machine 2 expansipon valf pid
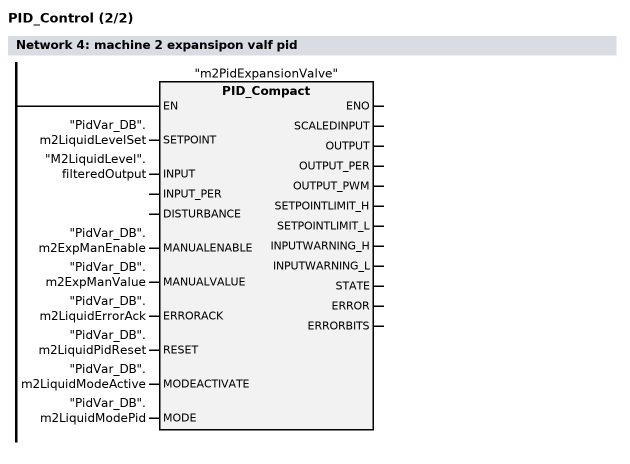
   "m2PidExpansionValve"(Setpoint := "PidVar_DB".m2LiquidLevelSet,   // PID_Compact
                         Input := "M2LiquidLevel".filteredOutput,
                         ManualEnable := "PidVar_DB".m2ExpManEnable,
                         ManualValue := "PidVar_DB".m2ExpManValue,
                         ErrorAck := "PidVar_DB".m2LiquidErrorAck,
                         Reset := "PidVar_DB".m2LiquidPidReset,
                         ModeActivate := "PidVar_DB".m2LiquidModeActive,
                         Mode := "PidVar_DB".m2LiquidModePid);
END_REGION
END_ORGANIZATION_BLOCK